LIN {X 0,Y 552.271,Z 509.997,A -85,B 0,C 180,E1 25736.055,E2 25736.055} C_VEL
LIN {X 0,Y 552.344,Z 509.997,A -85,B 0,C 180,E1 25732.825,E2 25732.825} C_VEL
LIN {X 0,Y 552.282,Z 509.996,A -85,B 0,C 180,E1 25729.569,E2 25729.569} C_VEL
LIN {X 0,Y 552.302,Z 509.994,A -85,B 0,C 180,E1 25726.174,E2 25726.174} C_VEL
LIN {X 0,Y 552.314,Z 509.999,A -85,B 0,C 180,E1 25723.054,E2 25723.054} C_VEL
LIN {X 0,Y 552.293,Z 509.995,A -85,B 0,C 180,E1 25719.77,E2 25719.77} C_VEL
LIN {X 0,Y 552.346,Z 509.995,A -85,B 0,C 180,E1 25716.531,E2 25716.531} C_VEL
LIN {X 0,Y 552.294,Z 509.997,A -85,B 0,C 180,E1 25713.322,E2 25713.322} C_VEL
LIN {X 0,Y 552.334,Z 509.997,A -85,B 0,C 180,E1 25712.64,E2 25712.64} C_VEL
LIN {X 0,Y 551.383,Z 510.118,A -85,B 0,C 180,E1 25711.84,E2 25711.84} C_VEL
LIN {X 0,Y 544.892,Z 510.92,A -85,B 0,C 180,E1 25709.597,E2 25709.597} C_VEL
LIN {X 0,Y 544.366,Z 510.988,A -85,B 0,C 180,E1 25709.012,E2 25709.012} C_VEL
LIN {X 0,Y 544.378,Z 510.984,A -85,B 0,C 180,E1 25705.546,E2 25705.546} C_VEL
LIN {X 0,Y 544.404,Z 510.987,A -85,B 0,C 180,E1 25702.162,E2 25702.162} C_VEL
LIN {X 0,Y 544.392,Z 511.152,A -85,B 0,C 180,E1 25698.937,E2 25698.937} C_VEL
LIN {X 0,Y 547.447,Z 523.021,A -85,B 0,C 180,E1 25697.272,E2 25697.272} C_VEL
LIN {X 0,Y 546.534,Z 551.773,A -85,B 0,C 180,E1 25693.828,E2 25693.828} C_VEL
LIN {X 0,Y 545.828,Z 580.978,A -85,B 0,C 180,E1 25690.42,E2 25690.42} C_VEL
LIN {X 0,Y 545.2,Z 610.398,A -85,B 0,C 180,E1 25687.05,E2 25687.05} C_VEL
LIN {X 0,Y 544.844,Z 632.663,A -85,B 0,C 180,E1 25684.588,E2 25684.588} C_VEL
LIN {X 0,Y 545.702,Z 641.313,A -85,B 0,C 180,E1 25684.418,E2 25684.418} C_VEL
LIN {X 0,Y 545.321,Z 744.483,A -85,B 0,C 180,E1 25683.029,E2 25683.029} C_VEL
LIN {X 0,Y 545.211,Z 758.833,A -85,B 0,C 180,E1 25682.65,E2 25682.65} C_VEL
LIN {X 0,Y 545.008,Z 773.495,A -85,B 0,C 180,E1 25682.051,E2 25682.051} C_VEL
LIN {X 0,Y 544.775,Z 786.249,A -85,B 0,C 180,E1 25681.334,E2 25681.334} C_VEL
LIN {X 0,Y 544.529,Z 799.172,A -85,B 0,C 180,E1 25680.385,E2 25680.385} C_VEL
LIN {X 0,Y 544.328,Z 811.081,A -85,B 0,C 180,E1 25679.245,E2 25679.245} C_VEL
LIN {X 0,Y 544.163,Z 820.825,A -85,B 0,C 180,E1 25678.055,E2 25678.055} C_VEL
LIN {X 0,Y 544.035,Z 829.383,A -85,B 0,C 180,E1 25676.721,E2 25676.721} C_VEL
LIN {X 0,Y 543.965,Z 836.569,A -85,B 0,C 180,E1 25675.238,E2 25675.238} C_VEL
LIN {X 0,Y 543.929,Z 841.752,A -85,B 0,C 180,E1 25673.732,E2 25673.732} C_VEL
LIN {X 0,Y 543.919,Z 845.089,A -85,B 0,C 180,E1 25672.248,E2 25672.248} C_VEL
LIN {X 0,Y 543.918,Z 846.806,A -85,B 0,C 180,E1 25670.662,E2 25670.662} C_VEL
LIN {X 0,Y 543.915,Z 846.71,A -85,B 0,C 180,E1 25669.096,E2 25669.096} C_VEL
LIN {X 0,Y 543.919,Z 844.892,A -85,B 0,C 180,E1 25667.543,E2 25667.543} C_VEL
LIN {X 0,Y 543.934,Z 840.933,A -85,B 0,C 180,E1 25665.893,E2 25665.893} C_VEL
LIN {X 0,Y 543.977,Z 835.236,A -85,B 0,C 180,E1 25664.365,E2 25664.365} C_VEL
LIN {X 0,Y 544.044,Z 828.675,A -85,B 0,C 180,E1 25663.062,E2 25663.062} C_VEL
LIN {X 0,Y 544.186,Z 819.39,A -85,B 0,C 180,E1 25661.658,E2 25661.658} C_VEL
LIN {X 0,Y 544.369,Z 808.765,A -85,B 0,C 180,E1 25660.421,E2 25660.421} C_VEL
LIN {X 0,Y 544.567,Z 797.66,A -85,B 0,C 180,E1 25659.403,E2 25659.403} C_VEL
LIN {X 0,Y 544.807,Z 784.989,A -85,B 0,C 180,E1 25658.494,E2 25658.494} C_VEL
LIN {X 0,Y 545.046,Z 771.112,A -85,B 0,C 180,E1 25657.747,E2 25657.747} C_VEL
LIN {X 0,Y 545.236,Z 756.981,A -85,B 0,C 180,E1 25657.202,E2 25657.202} C_VEL
LIN {X 0,Y 545.376,Z 741.93,A -85,B 0,C 180,E1 25656.832,E2 25656.832} C_VEL
LIN {X 0,Y 545.48,Z 637.399,A -85,B 0,C 180,E1 25655.434,E2 25655.434} C_VEL
LIN {X 0,Y 544.882,Z 632.555,A -85,B 0,C 180,E1 25655.315,E2 25655.315} C_VEL
LIN {X 0,Y 545.289,Z 602.715,A -85,B 0,C 180,E1 25651.995,E2 25651.995} C_VEL
LIN {X 0,Y 545.985,Z 572.64,A -85,B 0,C 180,E1 25648.53,E2 25648.53} C_VEL
LIN {X 0,Y 546.649,Z 544.661,A -85,B 0,C 180,E1 25645.278,E2 25645.278} C_VEL
LIN {X 0,Y 547.279,Z 522.265,A -85,B 0,C 180,E1 25642.599,E2 25642.599} C_VEL
LIN {X 0,Y 544.347,Z 511.079,A -85,B 0,C 180,E1 25640.991,E2 25640.991} C_VEL
LIN {X 0,Y 544.371,Z 510.988,A -85,B 0,C 180,E1 25637.806,E2 25637.806} C_VEL
LIN {X 0,Y 544.322,Z 510.99,A -85,B 0,C 180,E1 25634.553,E2 25634.553} C_VEL
LIN {X 0,Y 544.393,Z 510.99,A -85,B 0,C 180,E1 25631.363,E2 25631.363} C_VEL
LIN {X 0,Y 544.318,Z 510.989,A -85,B 0,C 180,E1 25628.22,E2 25628.22} C_VEL
LIN {X 0,Y 544.379,Z 510.983,A -85,B 0,C 180,E1 25625.012,E2 25625.012} C_VEL
LIN {X 0,Y 544.319,Z 510.989,A -85,B 0,C 180,E1 25621.832,E2 25621.832} C_VEL
LIN {X 0,Y 544.334,Z 510.982,A -85,B 0,C 180,E1 25618.434,E2 25618.434} C_VEL
LIN {X 0,Y 544.336,Z 510.989,A -85,B 0,C 180,E1 25615.377,E2 25615.377} C_VEL
LIN {X 0,Y 544.323,Z 510.987,A -85,B 0,C 180,E1 25612.002,E2 25612.002} C_VEL
LIN {X 0,Y 544.354,Z 510.99,A -85,B 0,C 180,E1 25609.019,E2 25609.019} C_VEL
LIN {X 0,Y 544.323,Z 510.988,A -85,B 0,C 180,E1 25605.735,E2 25605.735} C_VEL
LIN {X 0,Y 544.393,Z 510.985,A -85,B 0,C 180,E1 25602.524,E2 25602.524} C_VEL
LIN {X 0,Y 544.325,Z 510.986,A -85,B 0,C 180,E1 25599.326,E2 25599.326} C_VEL
LIN {X 0,Y 544.383,Z 510.983,A -85,B 0,C 180,E1 25596.09,E2 25596.09} C_VEL
LIN {X 0,Y 544.33,Z 510.982,A -85,B 0,C 180,E1 25592.937,E2 25592.937} C_VEL
LIN {X 0,Y 544.353,Z 510.986,A -85,B 0,C 180,E1 25589.61,E2 25589.61} C_VEL
LIN {X 0,Y 544.346,Z 510.982,A -85,B 0,C 180,E1 25586.56,E2 25586.56} C_VEL
LIN {X 0,Y 544.338,Z 510.986,A -85,B 0,C 180,E1 25583.147,E2 25583.147} C_VEL
LIN {X 0,Y 544.386,Z 510.988,A -85,B 0,C 180,E1 25579.976,E2 25579.976} C_VEL
LIN {X 0,Y 544.334,Z 510.979,A -85,B 0,C 180,E1 25576.762,E2 25576.762} C_VEL
LIN {X 0,Y 544.404,Z 510.987,A -85,B 0,C 180,E1 25573.597,E2 25573.597} C_VEL
LIN {X 0,Y 544.338,Z 510.983,A -85,B 0,C 180,E1 25570.371,E2 25570.371} C_VEL
LIN {X 0,Y 544.381,Z 510.981,A -85,B 0,C 180,E1 25567.069,E2 25567.069} C_VEL
LIN {X 0,Y 544.355,Z 510.987,A -85,B 0,C 180,E1 25563.897,E2 25563.897} C_VEL
LIN {X 0,Y 544.346,Z 510.974,A -85,B 0,C 180,E1 25560.421,E2 25560.421} C_VEL
LIN {X 0,Y 544.403,Z 510.988,A -85,B 0,C 180,E1 25557.158,E2 25557.158} C_VEL
LIN {X 0,Y 544.345,Z 510.984,A -85,B 0,C 180,E1 25553.885,E2 25553.885} C_VEL
LIN {X 0,Y 544.39,Z 510.982,A -85,B 0,C 180,E1 25550.592,E2 25550.592} C_VEL
LIN {X 0,Y 544.362,Z 510.987,A -85,B 0,C 180,E1 25547.375,E2 25547.375} C_VEL
LIN {X 0,Y 544.36,Z 510.981,A -85,B 0,C 180,E1 25544.008,E2 25544.008} C_VEL
LIN {X 0,Y 544.402,Z 510.985,A -85,B 0,C 180,E1 25540.728,E2 25540.728} C_VEL
LIN {X 0,Y 544.351,Z 510.984,A -85,B 0,C 180,E1 25537.425,E2 25537.425} C_VEL
LIN {X 0,Y 544.394,Z 510.977,A -85,B 0,C 180,E1 25534.08,E2 25534.08} C_VEL
LIN {X 0,Y 544.369,Z 510.987,A -85,B 0,C 180,E1 25530.874,E2 25530.874} C_VEL
LIN {X 0,Y 544.363,Z 510.983,A -85,B 0,C 180,E1 25527.441,E2 25527.441} C_VEL
LIN {X 0,Y 544.406,Z 510.985,A -85,B 0,C 180,E1 25524.135,E2 25524.135} C_VEL
LIN {X 0,Y 544.361,Z 510.984,A -85,B 0,C 180,E1 25520.811,E2 25520.811} C_VEL
LIN {X 0,Y 544.388,Z 510.982,A -85,B 0,C 180,E1 25517.431,E2 25517.431} C_VEL
LIN {X 0,Y 544.396,Z 510.987,A -85,B 0,C 180,E1 25514.1,E2 25514.1} C_VEL
LIN {X 0,Y 544.365,Z 510.985,A -85,B 0,C 180,E1 25510.823,E2 25510.823} C_VEL
LIN {X 0,Y 544.403,Z 510.987,A -85,B 0,C 180,E1 25507.57,E2 25507.57} C_VEL
LIN {X 0,Y 544.373,Z 510.989,A -85,B 0,C 180,E1 25504.195,E2 25504.195} C_VEL
LIN {X 0,Y 544.422,Z 511.233,A -85,B 0,C 180,E1 25502.897,E2 25502.897} C_VEL
LIN {X 0,Y 549.604,Z 527.102,A -85,B 0,C 180,E1 25501.29,E2 25501.29} C_VEL
LIN {X 0,Y 548.716,Z 570.56,A -85,B 0,C 180,E1 25498.124,E2 25498.124} C_VEL
LIN {X 0,Y 547.856,Z 611.744,A -85,B 0,C 180,E1 25495.147,E2 25495.147} C_VEL
LIN {X 0,Y 547.921,Z 615.465,A -85,B 0,C 180,E1 25494.922,E2 25494.922} C_VEL
LIN {X 0,Y 549.114,Z 624.911,A -85,B 0,C 180,E1 25494.729,E2 25494.729} C_VEL
LIN {X 0,Y 547.999,Z 824.349,A -85,B 0,C 180,E1 25491.964,E2 25491.964} C_VEL
LIN {X 0,Y 547.675,Z 843.385,A -85,B 0,C 180,E1 25491.502,E2 25491.502} C_VEL
LIN {X 0,Y 547.289,Z 861.41,A -85,B 0,C 180,E1 25490.87,E2 25490.87} C_VEL
LIN {X 0,Y 546.826,Z 879.05,A -85,B 0,C 180,E1 25490.049,E2 25490.049} C_VEL
LIN {X 0,Y 546.332,Z 895.775,A -85,B 0,C 180,E1 25489.067,E2 25489.067} C_VEL
LIN {X 0,Y 545.854,Z 911.628,A -85,B 0,C 180,E1 25487.922,E2 25487.922} C_VEL
LIN {X 0,Y 545.377,Z 926.557,A -85,B 0,C 180,E1 25486.618,E2 25486.618} C_VEL
LIN {X 0,Y 544.959,Z 940.217,A -85,B 0,C 180,E1 25485.187,E2 25485.187} C_VEL
LIN {X 0,Y 544.601,Z 952.914,A -85,B 0,C 180,E1 25483.592,E2 25483.592} C_VEL
LIN {X 0,Y 544.329,Z 964.228,A -85,B 0,C 180,E1 25481.872,E2 25481.872} C_VEL
LIN {X 0,Y 544.129,Z 973.992,A -85,B 0,C 180,E1 25480.054,E2 25480.054} C_VEL
LIN {X 0,Y 544.005,Z 982.175,A -85,B 0,C 180,E1 25478.137,E2 25478.137} C_VEL
LIN {X 0,Y 543.947,Z 988.41,A -85,B 0,C 180,E1 25476.227,E2 25476.227} C_VEL
LIN {X 0,Y 543.923,Z 992.876,A -85,B 0,C 180,E1 25474.323,E2 25474.323} C_VEL
LIN {X 0,Y 543.914,Z 995.792,A -85,B 0,C 180,E1 25472.319,E2 25472.319} C_VEL
LIN {X 0,Y 543.908,Z 996.939,A -85,B 0,C 180,E1 25470.317,E2 25470.317} C_VEL
LIN {X 0,Y 543.913,Z 996.348,A -85,B 0,C 180,E1 25468.316,E2 25468.316} C_VEL
LIN {X 0,Y 543.915,Z 994.005,A -85,B 0,C 180,E1 25466.313,E2 25466.313} C_VEL
LIN {X 0,Y 543.931,Z 990.101,A -85,B 0,C 180,E1 25464.411,E2 25464.411} C_VEL
LIN {X 0,Y 543.981,Z 984.474,A -85,B 0,C 180,E1 25462.503,E2 25462.503} C_VEL
LIN {X 0,Y 544.075,Z 977.436,A -85,B 0,C 180,E1 25460.695,E2 25460.695} C_VEL
LIN {X 0,Y 544.235,Z 968.529,A -85,B 0,C 180,E1 25458.88,E2 25458.88} C_VEL
LIN {X 0,Y 544.471,Z 958.168,A -85,B 0,C 180,E1 25457.164,E2 25457.164} C_VEL
LIN {X 0,Y 544.779,Z 946.371,A -85,B 0,C 180,E1 25455.548,E2 25455.548} C_VEL
LIN {X 0,Y 545.179,Z 933.106,A -85,B 0,C 180,E1 25454.035,E2 25454.035} C_VEL
LIN {X 0,Y 545.648,Z 918.253,A -85,B 0,C 180,E1 25452.624,E2 25452.624} C_VEL
LIN {X 0,Y 546.157,Z 902.275,A -85,B 0,C 180,E1 25451.373,E2 25451.373} C_VEL
LIN {X 0,Y 546.64,Z 885.106,A -85,B 0,C 180,E1 25450.28,E2 25450.28} C_VEL
LIN {X 0,Y 547.135,Z 867.88,A -85,B 0,C 180,E1 25449.407,E2 25449.407} C_VEL
LIN {X 0,Y 547.54,Z 849.631,A -85,B 0,C 180,E1 25448.695,E2 25448.695} C_VEL
LIN {X 0,Y 547.894,Z 830.962,A -85,B 0,C 180,E1 25448.175,E2 25448.175} C_VEL
LIN {X 0,Y 548.115,Z 810.606,A -85,B 0,C 180,E1 25447.822,E2 25447.822} C_VEL
LIN {X 0,Y 548.944,Z 622.019,A -85,B 0,C 180,E1 25445.222,E2 25445.222} C_VEL
LIN {X 0,Y 547.815,Z 614.387,A -85,B 0,C 180,E1 25445.038,E2 25445.038} C_VEL
LIN {X 0,Y 548.696,Z 571.729,A -85,B 0,C 180,E1 25441.961,E2 25441.961} C_VEL
LIN {X 0,Y 549.586,Z 527.86,A -85,B 0,C 180,E1 25438.767,E2 25438.767} C_VEL
LIN {X 0,Y 549.189,Z 525.155,A -85,B 0,C 180,E1 25438.534,E2 25438.534} C_VEL
LIN {X 0,Y 544.419,Z 511.228,A -85,B 0,C 180,E1 25437.106,E2 25437.106} C_VEL
LIN {X 0,Y 544.367,Z 510.99,A -85,B 0,C 180,E1 25433.739,E2 25433.739} C_VEL
LIN {X 0,Y 544.406,Z 510.984,A -85,B 0,C 180,E1 25430.415,E2 25430.415} C_VEL
LIN {X 0,Y 544.358,Z 510.985,A -85,B 0,C 180,E1 25427.127,E2 25427.127} C_VEL
LIN {X 0,Y 544.38,Z 510.99,A -85,B 0,C 180,E1 25423.802,E2 25423.802} C_VEL
LIN {X 0,Y 544.386,Z 510.984,A -85,B 0,C 180,E1 25420.51,E2 25420.51} C_VEL
LIN {X 0,Y 544.345,Z 510.988,A -85,B 0,C 180,E1 25417.148,E2 25417.148} C_VEL
LIN {X 0,Y 544.402,Z 510.987,A -85,B 0,C 180,E1 25413.896,E2 25413.896} C_VEL
LIN {X 0,Y 544.341,Z 510.986,A -85,B 0,C 180,E1 25410.706,E2 25410.706} C_VEL
LIN {X 0,Y 544.359,Z 510.988,A -85,B 0,C 180,E1 25407.335,E2 25407.335} C_VEL
LIN {X 0,Y 544.355,Z 510.986,A -85,B 0,C 180,E1 25404.18,E2 25404.18} C_VEL
LIN {X 0,Y 544.331,Z 510.988,A -85,B 0,C 180,E1 25400.876,E2 25400.876} C_VEL
LIN {X 0,Y 544.39,Z 510.985,A -85,B 0,C 180,E1 25397.641,E2 25397.641} C_VEL
LIN {X 0,Y 544.317,Z 510.983,A -85,B 0,C 180,E1 25394.467,E2 25394.467} C_VEL
LIN {X 0,Y 544.377,Z 510.987,A -85,B 0,C 180,E1 25391.226,E2 25391.226} C_VEL
LIN {X 0,Y 544.324,Z 510.988,A -85,B 0,C 180,E1 25388.025,E2 25388.025} C_VEL
LIN {X 0,Y 544.338,Z 510.984,A -85,B 0,C 180,E1 25384.636,E2 25384.636} C_VEL
LIN {X 0,Y 544.35,Z 510.989,A -85,B 0,C 180,E1 25381.579,E2 25381.579} C_VEL
LIN {X 0,Y 544.333,Z 510.987,A -85,B 0,C 180,E1 25378.21,E2 25378.21} C_VEL
LIN {X 0,Y 544.399,Z 510.982,A -85,B 0,C 180,E1 25374.942,E2 25374.942} C_VEL
LIN {X 0,Y 544.337,Z 510.987,A -85,B 0,C 180,E1 25371.762,E2 25371.762} C_VEL
LIN {X 0,Y 544.383,Z 510.985,A -85,B 0,C 180,E1 25368.451,E2 25368.451} C_VEL
LIN {X 0,Y 544.355,Z 510.985,A -85,B 0,C 180,E1 25365.316,E2 25365.316} C_VEL
LIN {X 0,Y 544.358,Z 510.984,A -85,B 0,C 180,E1 25361.916,E2 25361.916} C_VEL
LIN {X 0,Y 544.405,Z 510.984,A -85,B 0,C 180,E1 25358.6,E2 25358.6} C_VEL
LIN {X 0,Y 544.353,Z 510.983,A -85,B 0,C 180,E1 25355.358,E2 25355.358} C_VEL
LIN {X 0,Y 544.404,Z 510.983,A -85,B 0,C 180,E1 25352.044,E2 25352.044} C_VEL
LIN {X 0,Y 544.366,Z 510.988,A -85,B 0,C 180,E1 25349.012,E2 25349.012} C_VEL
LIN {X 0,Y 543.401,Z 511.113,A -85,B 0,C 180,E1 25348.201,E2 25348.201} C_VEL
LIN {X 0,Y 536.881,Z 511.92,A -85,B 0,C 180,E1 25345.865,E2 25345.865} C_VEL
LIN {X 0,Y 536.428,Z 511.975,A -85,B 0,C 180,E1 25345.33,E2 25345.33} C_VEL
LIN {X 0,Y 536.464,Z 511.977,A -85,B 0,C 180,E1 25342.026,E2 25342.026} C_VEL
LIN {X 0,Y 536.478,Z 512.244,A -85,B 0,C 180,E1 25339.304,E2 25339.304} C_VEL
LIN {X 0,Y 539.943,Z 525.069,A -85,B 0,C 180,E1 25337.47,E2 25337.47} C_VEL
LIN {X 0,Y 538.944,Z 553.767,A -85,B 0,C 180,E1 25333.996,E2 25333.996} C_VEL
LIN {X 0,Y 538.16,Z 583.042,A -85,B 0,C 180,E1 25330.545,E2 25330.545} C_VEL
LIN {X 0,Y 537.38,Z 612.981,A -85,B 0,C 180,E1 25327.04,E2 25327.04} C_VEL
LIN {X 0,Y 536.989,Z 632.746,A -85,B 0,C 180,E1 25324.801,E2 25324.801} C_VEL
LIN {X 0,Y 537.953,Z 642.099,A -85,B 0,C 180,E1 25324.62,E2 25324.62} C_VEL
LIN {X 0,Y 537.526,Z 744.402,A -85,B 0,C 180,E1 25323.223,E2 25323.223} C_VEL
LIN {X 0,Y 537.391,Z 759.339,A -85,B 0,C 180,E1 25322.821,E2 25322.821} C_VEL
LIN {X 0,Y 537.159,Z 774.098,A -85,B 0,C 180,E1 25322.201,E2 25322.201} C_VEL
LIN {X 0,Y 536.878,Z 787.415,A -85,B 0,C 180,E1 25321.426,E2 25321.426} C_VEL
LIN {X 0,Y 536.618,Z 799.477,A -85,B 0,C 180,E1 25320.513,E2 25320.513} C_VEL
LIN {X 0,Y 536.387,Z 811.37,A -85,B 0,C 180,E1 25319.353,E2 25319.353} C_VEL
LIN {X 0,Y 536.194,Z 821.279,A -85,B 0,C 180,E1 25318.112,E2 25318.112} C_VEL
LIN {X 0,Y 536.056,Z 829.352,A -85,B 0,C 180,E1 25316.828,E2 25316.828} C_VEL
LIN {X 0,Y 535.971,Z 836.696,A -85,B 0,C 180,E1 25315.286,E2 25315.286} C_VEL
LIN {X 0,Y 535.931,Z 841.829,A -85,B 0,C 180,E1 25313.761,E2 25313.761} C_VEL
LIN {X 0,Y 535.919,Z 845.135,A -85,B 0,C 180,E1 25312.252,E2 25312.252} C_VEL
LIN {X 0,Y 535.918,Z 846.824,A -85,B 0,C 180,E1 25310.644,E2 25310.644} C_VEL
LIN {X 0,Y 535.915,Z 846.691,A -85,B 0,C 180,E1 25309.053,E2 25309.053} C_VEL
LIN {X 0,Y 535.919,Z 844.836,A -85,B 0,C 180,E1 25307.477,E2 25307.477} C_VEL
LIN {X 0,Y 535.938,Z 840.849,A -85,B 0,C 180,E1 25305.803,E2 25305.803} C_VEL
LIN {X 0,Y 535.987,Z 835.114,A -85,B 0,C 180,E1 25304.252,E2 25304.252} C_VEL
LIN {X 0,Y 536.08,Z 827.859,A -85,B 0,C 180,E1 25302.821,E2 25302.821} C_VEL
LIN {X 0,Y 536.235,Z 819.186,A -85,B 0,C 180,E1 25301.506,E2 25301.506} C_VEL
LIN {X 0,Y 536.452,Z 808.273,A -85,B 0,C 180,E1 25300.227,E2 25300.227} C_VEL
LIN {X 0,Y 536.682,Z 796.645,A -85,B 0,C 180,E1 25299.164,E2 25299.164} C_VEL
LIN {X 0,Y 536.952,Z 784.539,A -85,B 0,C 180,E1 25298.295,E2 25298.295} C_VEL
LIN {X 0,Y 537.22,Z 770.517,A -85,B 0,C 180,E1 25297.538,E2 25297.538} C_VEL
LIN {X 0,Y 537.439,Z 756.126,A -85,B 0,C 180,E1 25296.987,E2 25296.987} C_VEL
LIN {X 0,Y 537.587,Z 741.359,A -85,B 0,C 180,E1 25296.629,E2 25296.629} C_VEL
LIN {X 0,Y 537.745,Z 638.26,A -85,B 0,C 180,E1 25295.232,E2 25295.232} C_VEL
LIN {X 0,Y 537.021,Z 632.585,A -85,B 0,C 180,E1 25295.099,E2 25295.099} C_VEL
LIN {X 0,Y 537.544,Z 603.794,A -85,B 0,C 180,E1 25291.811,E2 25291.811} C_VEL
LIN {X 0,Y 538.357,Z 572.84,A -85,B 0,C 180,E1 25288.19,E2 25288.19} C_VEL
LIN {X 0,Y 539.12,Z 544.837,A -85,B 0,C 180,E1 25284.892,E2 25284.892} C_VEL
LIN {X 0,Y 539.654,Z 524.364,A -85,B 0,C 180,E1 25282.412,E2 25282.412} C_VEL
LIN {X 0,Y 536.398,Z 512.075,A -85,B 0,C 180,E1 25280.613,E2 25280.613} C_VEL
LIN {X 0,Y 536.435,Z 511.979,A -85,B 0,C 180,E1 25277.294,E2 25277.294} C_VEL
LIN {X 0,Y 536.386,Z 511.979,A -85,B 0,C 180,E1 25274.208,E2 25274.208} C_VEL
LIN {X 0,Y 536.405,Z 511.977,A -85,B 0,C 180,E1 25270.849,E2 25270.849} C_VEL
LIN {X 0,Y 536.398,Z 511.978,A -85,B 0,C 180,E1 25267.766,E2 25267.766} C_VEL
LIN {X 0,Y 536.383,Z 511.978,A -85,B 0,C 180,E1 25264.377,E2 25264.377} C_VEL
LIN {X 0,Y 536.443,Z 511.969,A -85,B 0,C 180,E1 25261.137,E2 25261.137} C_VEL
LIN {X 0,Y 536.374,Z 511.97,A -85,B 0,C 180,E1 25257.91,E2 25257.91} C_VEL
LIN {X 0,Y 536.438,Z 511.977,A -85,B 0,C 180,E1 25254.706,E2 25254.706} C_VEL
LIN {X 0,Y 536.385,Z 511.976,A -85,B 0,C 180,E1 25251.496,E2 25251.496} C_VEL
LIN {X 0,Y 536.396,Z 511.972,A -85,B 0,C 180,E1 25248.052,E2 25248.052} C_VEL
LIN {X 0,Y 536.416,Z 511.977,A -85,B 0,C 180,E1 25244.906,E2 25244.906} C_VEL
LIN {X 0,Y 536.385,Z 511.97,A -85,B 0,C 180,E1 25241.576,E2 25241.576} C_VEL
LIN {X 0,Y 536.461,Z 511.977,A -85,B 0,C 180,E1 25238.364,E2 25238.364} C_VEL
LIN {X 0,Y 536.388,Z 511.973,A -85,B 0,C 180,E1 25235.088,E2 25235.088} C_VEL
LIN {X 0,Y 536.418,Z 511.975,A -85,B 0,C 180,E1 25231.711,E2 25231.711} C_VEL
LIN {X 0,Y 536.405,Z 511.977,A -85,B 0,C 180,E1 25228.624,E2 25228.624} C_VEL
LIN {X 0,Y 536.396,Z 511.969,A -85,B 0,C 180,E1 25225.151,E2 25225.151} C_VEL
LIN {X 0,Y 536.465,Z 511.977,A -85,B 0,C 180,E1 25221.886,E2 25221.886} C_VEL
LIN {X 0,Y 536.396,Z 511.97,A -85,B 0,C 180,E1 25218.588,E2 25218.588} C_VEL
LIN {X 0,Y 536.428,Z 511.973,A -85,B 0,C 180,E1 25215.237,E2 25215.237} C_VEL
LIN {X 0,Y 536.418,Z 511.977,A -85,B 0,C 180,E1 25212.05,E2 25212.05} C_VEL
LIN {X 0,Y 536.405,Z 511.963,A -85,B 0,C 180,E1 25208.684,E2 25208.684} C_VEL
LIN {X 0,Y 536.46,Z 511.976,A -85,B 0,C 180,E1 25205.455,E2 25205.455} C_VEL
LIN {X 0,Y 536.403,Z 511.972,A -85,B 0,C 180,E1 25202.137,E2 25202.137} C_VEL
LIN {X 0,Y 536.447,Z 511.97,A -85,B 0,C 180,E1 25198.825,E2 25198.825} C_VEL
LIN {X 0,Y 536.42,Z 511.977,A -85,B 0,C 180,E1 25195.617,E2 25195.617} C_VEL
LIN {X 0,Y 536.412,Z 511.965,A -85,B 0,C 180,E1 25192.18,E2 25192.18} C_VEL
LIN {X 0,Y 536.464,Z 511.977,A -85,B 0,C 180,E1 25188.932,E2 25188.932} C_VEL
LIN {X 0,Y 536.411,Z 511.969,A -85,B 0,C 180,E1 25185.646,E2 25185.646} C_VEL
LIN {X 0,Y 536.453,Z 511.972,A -85,B 0,C 180,E1 25182.314,E2 25182.314} C_VEL
LIN {X 0,Y 536.433,Z 511.973,A -85,B 0,C 180,E1 25179.028,E2 25179.028} C_VEL
LIN {X 0,Y 536.42,Z 511.973,A -85,B 0,C 180,E1 25175.674,E2 25175.674} C_VEL
LIN {X 0,Y 536.468,Z 511.974,A -85,B 0,C 180,E1 25172.349,E2 25172.349} C_VEL
LIN {X 0,Y 536.421,Z 511.973,A -85,B 0,C 180,E1 25169.022,E2 25169.022} C_VEL
LIN {X 0,Y 536.439,Z 511.97,A -85,B 0,C 180,E1 25165.615,E2 25165.615} C_VEL
LIN {X 0,Y 536.46,Z 511.978,A -85,B 0,C 180,E1 25162.314,E2 25162.314} C_VEL
LIN {X 0,Y 536.422,Z 511.974,A -85,B 0,C 180,E1 25158.996,E2 25158.996} C_VEL
LIN {X 0,Y 536.465,Z 511.969,A -85,B 0,C 180,E1 25155.66,E2 25155.66} C_VEL
LIN {X 0,Y 536.439,Z 511.976,A -85,B 0,C 180,E1 25152.272,E2 25152.272} C_VEL
LIN {X 0,Y 536.43,Z 511.974,A -85,B 0,C 180,E1 25148.82,E2 25148.82} C_VEL
LIN {X 0,Y 536.464,Z 511.973,A -85,B 0,C 180,E1 25145.423,E2 25145.423} C_VEL
LIN {X 0,Y 536.497,Z 512.203,A -85,B 0,C 180,E1 25143.331,E2 25143.331} C_VEL
LIN {X 0,Y 542.287,Z 529.764,A -85,B 0,C 180,E1 25141.513,E2 25141.513} C_VEL
LIN {X 0,Y 541.221,Z 573.376,A -85,B 0,C 180,E1 25138.284,E2 25138.284} C_VEL
LIN {X 0,Y 540.42,Z 615.037,A -85,B 0,C 180,E1 25135.298,E2 25135.298} C_VEL
LIN {X 0,Y 541.842,Z 625.928,A -85,B 0,C 180,E1 25135.069,E2 25135.069} C_VEL
LIN {X 0,Y 540.578,Z 824.349,A -85,B 0,C 180,E1 25132.282,E2 25132.282} C_VEL
LIN {X 0,Y 540.217,Z 843.359,A -85,B 0,C 180,E1 25131.815,E2 25131.815} C_VEL
LIN {X 0,Y 539.775,Z 861.408,A -85,B 0,C 180,E1 25131.174,E2 25131.174} C_VEL
LIN {X 0,Y 539.254,Z 879.047,A -85,B 0,C 180,E1 25130.343,E2 25130.343} C_VEL
LIN {X 0,Y 538.689,Z 895.773,A -85,B 0,C 180,E1 25129.348,E2 25129.348} C_VEL
LIN {X 0,Y 538.124,Z 912.195,A -85,B 0,C 180,E1 25128.141,E2 25128.141} C_VEL
LIN {X 0,Y 537.582,Z 927.111,A -85,B 0,C 180,E1 25126.811,E2 25126.811} C_VEL
LIN {X 0,Y 537.097,Z 940.945,A -85,B 0,C 180,E1 25125.328,E2 25125.328} C_VEL
LIN {X 0,Y 536.688,Z 953.683,A -85,B 0,C 180,E1 25123.686,E2 25123.686} C_VEL
LIN {X 0,Y 536.38,Z 964.863,A -85,B 0,C 180,E1 25121.942,E2 25121.942} C_VEL
LIN {X 0,Y 536.155,Z 974.506,A -85,B 0,C 180,E1 25120.096,E2 25120.096} C_VEL
LIN {X 0,Y 536.023,Z 982.174,A -85,B 0,C 180,E1 25118.259,E2 25118.259} C_VEL
LIN {X 0,Y 535.953,Z 988.411,A -85,B 0,C 180,E1 25116.32,E2 25116.32} C_VEL
LIN {X 0,Y 535.924,Z 992.876,A -85,B 0,C 180,E1 25114.388,E2 25114.388} C_VEL
LIN {X 0,Y 535.913,Z 995.792,A -85,B 0,C 180,E1 25112.354,E2 25112.354} C_VEL
LIN {X 0,Y 535.908,Z 996.939,A -85,B 0,C 180,E1 25110.322,E2 25110.322} C_VEL
LIN {X 0,Y 535.913,Z 996.348,A -85,B 0,C 180,E1 25108.291,E2 25108.291} C_VEL
LIN {X 0,Y 535.917,Z 994.004,A -85,B 0,C 180,E1 25106.258,E2 25106.258} C_VEL
LIN {X 0,Y 535.934,Z 990.101,A -85,B 0,C 180,E1 25104.327,E2 25104.327} C_VEL
LIN {X 0,Y 535.995,Z 984.474,A -85,B 0,C 180,E1 25102.391,E2 25102.391} C_VEL
LIN {X 0,Y 536.1,Z 977.436,A -85,B 0,C 180,E1 25100.556,E2 25100.556} C_VEL
LIN {X 0,Y 536.288,Z 968.53,A -85,B 0,C 180,E1 25098.713,E2 25098.713} C_VEL
LIN {X 0,Y 536.561,Z 958.169,A -85,B 0,C 180,E1 25096.971,E2 25096.971} C_VEL
LIN {X 0,Y 536.916,Z 946.371,A -85,B 0,C 180,E1 25095.332,E2 25095.332} C_VEL
LIN {X 0,Y 537.393,Z 932.684,A -85,B 0,C 180,E1 25093.751,E2 25093.751} C_VEL
LIN {X 0,Y 537.941,Z 917.637,A -85,B 0,C 180,E1 25092.311,E2 25092.311} C_VEL
LIN {X 0,Y 538.518,Z 901.481,A -85,B 0,C 180,E1 25091.042,E2 25091.042} C_VEL
LIN {X 0,Y 539.06,Z 884.78,A -85,B 0,C 180,E1 25089.973,E2 25089.973} C_VEL
LIN {X 0,Y 539.602,Z 867.882,A -85,B 0,C 180,E1 25089.106,E2 25089.106} C_VEL
LIN {X 0,Y 540.061,Z 849.634,A -85,B 0,C 180,E1 25088.385,E2 25088.385} C_VEL
LIN {X 0,Y 540.459,Z 831.074,A -85,B 0,C 180,E1 25087.861,E2 25087.861} C_VEL
LIN {X 0,Y 540.709,Z 810.733,A -85,B 0,C 180,E1 25087.503,E2 25087.503} C_VEL
LIN {X 0,Y 541.698,Z 623.241,A -85,B 0,C 180,E1 25084.885,E2 25084.885} C_VEL
LIN {X 0,Y 540.369,Z 614.302,A -85,B 0,C 180,E1 25084.67,E2 25084.67} C_VEL
LIN {X 0,Y 541.305,Z 569.367,A -85,B 0,C 180,E1 25081.423,E2 25081.423} C_VEL
LIN {X 0,Y 542.299,Z 529.19,A -85,B 0,C 180,E1 25078.445,E2 25078.445} C_VEL
LIN {X 0,Y 536.507,Z 512.263,A -85,B 0,C 180,E1 25076.688,E2 25076.688} C_VEL
LIN {X 0,Y 536.466,Z 511.975,A -85,B 0,C 180,E1 25074.58,E2 25074.58} C_VEL
LIN {X 0,Y 536.424,Z 511.974,A -85,B 0,C 180,E1 25071.229,E2 25071.229} C_VEL
LIN {X 0,Y 536.43,Z 511.977,A -85,B 0,C 180,E1 25067.729,E2 25067.729} C_VEL
LIN {X 0,Y 536.463,Z 511.973,A -85,B 0,C 180,E1 25064.459,E2 25064.459} C_VEL
LIN {X 0,Y 536.411,Z 511.975,A -85,B 0,C 180,E1 25061.146,E2 25061.146} C_VEL
LIN {X 0,Y 536.45,Z 511.978,A -85,B 0,C 180,E1 25057.798,E2 25057.798} C_VEL
LIN {X 0,Y 536.421,Z 511.973,A -85,B 0,C 180,E1 25054.516,E2 25054.516} C_VEL
LIN {X 0,Y 536.403,Z 511.976,A -85,B 0,C 180,E1 25051.086,E2 25051.086} C_VEL
LIN {X 0,Y 536.463,Z 511.97,A -85,B 0,C 180,E1 25047.892,E2 25047.892} C_VEL
LIN {X 0,Y 536.392,Z 511.975,A -85,B 0,C 180,E1 25044.68,E2 25044.68} C_VEL
LIN {X 0,Y 536.442,Z 511.978,A -85,B 0,C 180,E1 25041.427,E2 25041.427} C_VEL
LIN {X 0,Y 536.393,Z 511.974,A -85,B 0,C 180,E1 25038.25,E2 25038.25} C_VEL
LIN {X 0,Y 536.389,Z 511.971,A -85,B 0,C 180,E1 25034.796,E2 25034.796} C_VEL
LIN {X 0,Y 536.429,Z 511.979,A -85,B 0,C 180,E1 25031.613,E2 25031.613} C_VEL
LIN {X 0,Y 536.378,Z 511.977,A -85,B 0,C 180,E1 25028.36,E2 25028.36} C_VEL
LIN {X 0,Y 536.45,Z 511.97,A -85,B 0,C 180,E1 25025.133,E2 25025.133} C_VEL
LIN {X 0,Y 536.39,Z 511.978,A -85,B 0,C 180,E1 25021.923,E2 25021.923} C_VEL
LIN {X 0,Y 536.41,Z 511.976,A -85,B 0,C 180,E1 25018.504,E2 25018.504} C_VEL
LIN {X 0,Y 536.43,Z 511.975,A -85,B 0,C 180,E1 25015.296,E2 25015.296} C_VEL
LIN {X 0,Y 536.4,Z 511.976,A -85,B 0,C 180,E1 25011.963,E2 25011.963} C_VEL
LIN {X 0,Y 536.466,Z 511.975,A -85,B 0,C 180,E1 25008.714,E2 25008.714} C_VEL
LIN {X 0,Y 536.411,Z 511.974,A -85,B 0,C 180,E1 25005.425,E2 25005.425} C_VEL
LIN {X 0,Y 536.423,Z 511.972,A -85,B 0,C 180,E1 25001.976,E2 25001.976} C_VEL
LIN {X 0,Y 536.462,Z 511.973,A -85,B 0,C 180,E1 24998.688,E2 24998.688} C_VEL
LIN {X 0,Y 536.414,Z 511.972,A -85,B 0,C 180,E1 24995.438,E2 24995.438} C_VEL
LIN {X 0,Y 536.465,Z 511.972,A -85,B 0,C 180,E1 24992.048,E2 24992.048} C_VEL
LIN {X 0,Y 536.455,Z 511.977,A -85,B 0,C 180,E1 24988.598,E2 24988.598} C_VEL
LIN {X 0,Y 536.428,Z 511.975,A -85,B 0,C 180,E1 24985.33,E2 24985.33} C_VEL
LIN {X 0,Y 535.437,Z 512.103,A -85,B 0,C 180,E1 24984.508,E2 24984.508} C_VEL
LIN {X 0,Y 528.98,Z 512.908,A -85,B 0,C 180,E1 24982.136,E2 24982.136} C_VEL
LIN {X 0,Y 528.516,Z 512.964,A -85,B 0,C 180,E1 24981.594,E2 24981.594} C_VEL
LIN {X 0,Y 528.569,Z 513.247,A -85,B 0,C 180,E1 24979.711,E2 24979.711} C_VEL
LIN {X 0,Y 532.433,Z 527.639,A -85,B 0,C 180,E1 24977.61,E2 24977.61} C_VEL
LIN {X 0,Y 531.357,Z 556.238,A -85,B 0,C 180,E1 24974.119,E2 24974.119} C_VEL
LIN {X 0,Y 530.477,Z 585.499,A -85,B 0,C 180,E1 24970.627,E2 24970.627} C_VEL
LIN {X 0,Y 529.631,Z 614.708,A -85,B 0,C 180,E1 24967.159,E2 24967.159} C_VEL
LIN {X 0,Y 529.25,Z 632.819,A -85,B 0,C 180,E1 24965.088,E2 24965.088} C_VEL
LIN {X 0,Y 530.36,Z 642.793,A -85,B 0,C 180,E1 24964.883,E2 24964.883} C_VEL
LIN {X 0,Y 529.797,Z 744.646,A -85,B 0,C 180,E1 24963.443,E2 24963.443} C_VEL
LIN {X 0,Y 529.634,Z 758.971,A -85,B 0,C 180,E1 24963.049,E2 24963.049} C_VEL
LIN {X 0,Y 529.363,Z 773.363,A -85,B 0,C 180,E1 24962.435,E2 24962.435} C_VEL
LIN {X 0,Y 529.039,Z 786.603,A -85,B 0,C 180,E1 24961.657,E2 24961.657} C_VEL
LIN {X 0,Y 528.722,Z 799.187,A -85,B 0,C 180,E1 24960.699,E2 24960.699} C_VEL
LIN {X 0,Y 528.457,Z 811.32,A -85,B 0,C 180,E1 24959.501,E2 24959.501} C_VEL
LIN {X 0,Y 528.235,Z 821.262,A -85,B 0,C 180,E1 24958.238,E2 24958.238} C_VEL
LIN {X 0,Y 528.075,Z 829.526,A -85,B 0,C 180,E1 24956.9,E2 24956.9} C_VEL
LIN {X 0,Y 527.979,Z 836.819,A -85,B 0,C 180,E1 24955.336,E2 24955.336} C_VEL
LIN {X 0,Y 527.931,Z 842.245,A -85,B 0,C 180,E1 24953.669,E2 24953.669} C_VEL
LIN {X 0,Y 527.921,Z 845.526,A -85,B 0,C 180,E1 24952.021,E2 24952.021} C_VEL
LIN {X 0,Y 527.919,Z 846.889,A -85,B 0,C 180,E1 24950.507,E2 24950.507} C_VEL
LIN {X 0,Y 527.916,Z 846.528,A -85,B 0,C 180,E1 24948.779,E2 24948.779} C_VEL
LIN {X 0,Y 527.921,Z 844.348,A -85,B 0,C 180,E1 24947.182,E2 24947.182} C_VEL
LIN {X 0,Y 527.944,Z 840.405,A -85,B 0,C 180,E1 24945.598,E2 24945.598} C_VEL
LIN {X 0,Y 528.006,Z 834.519,A -85,B 0,C 180,E1 24944.025,E2 24944.025} C_VEL
LIN {X 0,Y 528.12,Z 827.044,A -85,B 0,C 180,E1 24942.573,E2 24942.573} C_VEL
LIN {X 0,Y 528.306,Z 818.121,A -85,B 0,C 180,E1 24941.239,E2 24941.239} C_VEL
LIN {X 0,Y 528.555,Z 807.188,A -85,B 0,C 180,E1 24939.965,E2 24939.965} C_VEL
LIN {X 0,Y 528.829,Z 794.954,A -85,B 0,C 180,E1 24938.862,E2 24938.862} C_VEL
LIN {X 0,Y 529.171,Z 781.448,A -85,B 0,C 180,E1 24937.926,E2 24937.926} C_VEL
LIN {X 0,Y 529.468,Z 768.133,A -85,B 0,C 180,E1 24937.229,E2 24937.229} C_VEL
LIN {X 0,Y 529.726,Z 753.411,A -85,B 0,C 180,E1 24936.688,E2 24936.688} C_VEL
LIN {X 0,Y 529.877,Z 737.548,A -85,B 0,C 180,E1 24936.346,E2 24936.346} C_VEL
LIN {X 0,Y 530.136,Z 639.111,A -85,B 0,C 180,E1 24934.975,E2 24934.975} C_VEL
LIN {X 0,Y 529.246,Z 632.589,A -85,B 0,C 180,E1 24934.821,E2 24934.821} C_VEL
LIN {X 0,Y 529.818,Z 604.948,A -85,B 0,C 180,E1 24931.621,E2 24931.621} C_VEL
LIN {X 0,Y 530.699,Z 574.865,A -85,B 0,C 180,E1 24928.055,E2 24928.055} C_VEL
LIN {X 0,Y 531.562,Z 546.856,A -85,B 0,C 180,E1 24924.711,E2 24924.711} C_VEL
LIN {X 0,Y 532.272,Z 527.363,A -85,B 0,C 180,E1 24922.335,E2 24922.335} C_VEL
LIN {X 0,Y 528.477,Z 513.102,A -85,B 0,C 180,E1 24920.251,E2 24920.251} C_VEL
LIN {X 0,Y 528.451,Z 512.967,A -85,B 0,C 180,E1 24916.765,E2 24916.765} C_VEL
LIN {X 0,Y 528.503,Z 512.968,A -85,B 0,C 180,E1 24913.574,E2 24913.574} C_VEL
LIN {X 0,Y 528.443,Z 512.966,A -85,B 0,C 180,E1 24910.319,E2 24910.319} C_VEL
LIN {X 0,Y 528.5,Z 512.949,A -85,B 0,C 180,E1 24907.063,E2 24907.063} C_VEL
LIN {X 0,Y 528.446,Z 512.967,A -85,B 0,C 180,E1 24903.843,E2 24903.843} C_VEL
LIN {X 0,Y 528.449,Z 512.952,A -85,B 0,C 180,E1 24900.409,E2 24900.409} C_VEL
LIN {X 0,Y 528.476,Z 512.958,A -85,B 0,C 180,E1 24897.243,E2 24897.243} C_VEL
LIN {X 0,Y 528.439,Z 512.966,A -85,B 0,C 180,E1 24893.894,E2 24893.894} C_VEL
LIN {X 0,Y 528.519,Z 512.967,A -85,B 0,C 180,E1 24890.675,E2 24890.675} C_VEL
LIN {X 0,Y 528.443,Z 512.96,A -85,B 0,C 180,E1 24887.512,E2 24887.512} C_VEL
LIN {X 0,Y 528.481,Z 512.966,A -85,B 0,C 180,E1 24884.192,E2 24884.192} C_VEL
LIN {X 0,Y 528.456,Z 512.959,A -85,B 0,C 180,E1 24881.037,E2 24881.037} C_VEL
LIN {X 0,Y 528.454,Z 512.966,A -85,B 0,C 180,E1 24877.559,E2 24877.559} C_VEL
LIN {X 0,Y 528.521,Z 512.954,A -85,B 0,C 180,E1 24874.242,E2 24874.242} C_VEL
LIN {X 0,Y 528.452,Z 512.965,A -85,B 0,C 180,E1 24870.974,E2 24870.974} C_VEL
LIN {X 0,Y 528.484,Z 512.957,A -85,B 0,C 180,E1 24867.615,E2 24867.615} C_VEL
LIN {X 0,Y 528.47,Z 512.959,A -85,B 0,C 180,E1 24864.478,E2 24864.478} C_VEL
LIN {X 0,Y 528.461,Z 512.964,A -85,B 0,C 180,E1 24861.069,E2 24861.069} C_VEL
LIN {X 0,Y 528.523,Z 512.952,A -85,B 0,C 180,E1 24857.733,E2 24857.733} C_VEL
LIN {X 0,Y 528.46,Z 512.964,A -85,B 0,C 180,E1 24854.463,E2 24854.463} C_VEL
LIN {X 0,Y 528.492,Z 512.958,A -85,B 0,C 180,E1 24851.127,E2 24851.127} C_VEL
LIN {X 0,Y 528.478,Z 512.953,A -85,B 0,C 180,E1 24847.939,E2 24847.939} C_VEL
LIN {X 0,Y 528.469,Z 512.963,A -85,B 0,C 180,E1 24844.558,E2 24844.558} C_VEL
LIN {X 0,Y 528.524,Z 512.952,A -85,B 0,C 180,E1 24841.301,E2 24841.301} C_VEL
LIN {X 0,Y 528.466,Z 512.961,A -85,B 0,C 180,E1 24838.049,E2 24838.049} C_VEL
LIN {X 0,Y 528.507,Z 512.958,A -85,B 0,C 180,E1 24834.681,E2 24834.681} C_VEL
LIN {X 0,Y 528.488,Z 512.956,A -85,B 0,C 180,E1 24831.404,E2 24831.404} C_VEL
LIN {X 0,Y 528.473,Z 512.963,A -85,B 0,C 180,E1 24827.984,E2 24827.984} C_VEL
LIN {X 0,Y 528.53,Z 512.957,A -85,B 0,C 180,E1 24824.642,E2 24824.642} C_VEL
LIN {X 0,Y 528.479,Z 512.965,A -85,B 0,C 180,E1 24821.353,E2 24821.353} C_VEL
LIN {X 0,Y 528.488,Z 512.959,A -85,B 0,C 180,E1 24817.884,E2 24817.884} C_VEL
LIN {X 0,Y 528.524,Z 512.96,A -85,B 0,C 180,E1 24814.568,E2 24814.568} C_VEL
LIN {X 0,Y 528.476,Z 512.964,A -85,B 0,C 180,E1 24811.278,E2 24811.278} C_VEL
LIN {X 0,Y 528.524,Z 512.959,A -85,B 0,C 180,E1 24807.938,E2 24807.938} C_VEL
LIN {X 0,Y 528.509,Z 512.962,A -85,B 0,C 180,E1 24804.493,E2 24804.493} C_VEL
LIN {X 0,Y 528.482,Z 512.96,A -85,B 0,C 180,E1 24801.088,E2 24801.088} C_VEL
LIN {X 0,Y 528.525,Z 512.961,A -85,B 0,C 180,E1 24797.811,E2 24797.811} C_VEL
LIN {X 0,Y 528.494,Z 512.963,A -85,B 0,C 180,E1 24794.424,E2 24794.424} C_VEL
LIN {X 0,Y 528.491,Z 512.963,A -85,B 0,C 180,E1 24790.887,E2 24790.887} C_VEL
LIN {X 0,Y 528.525,Z 512.965,A -85,B 0,C 180,E1 24787.526,E2 24787.526} C_VEL
LIN {X 0,Y 528.496,Z 512.968,A -85,B 0,C 180,E1 24784.185,E2 24784.185} C_VEL
LIN {X 0,Y 528.589,Z 513.411,A -85,B 0,C 180,E1 24783.733,E2 24783.733} C_VEL
LIN {X 0,Y 534.978,Z 532.365,A -85,B 0,C 180,E1 24781.747,E2 24781.747} C_VEL
LIN {X 0,Y 533.768,Z 574.446,A -85,B 0,C 180,E1 24778.578,E2 24778.578} C_VEL
LIN {X 0,Y 532.811,Z 615.221,A -85,B 0,C 180,E1 24775.598,E2 24775.598} C_VEL
LIN {X 0,Y 534.386,Z 626.877,A -85,B 0,C 180,E1 24775.368,E2 24775.368} C_VEL
LIN {X 0,Y 533.239,Z 818.243,A -85,B 0,C 180,E1 24772.713,E2 24772.713} C_VEL
LIN {X 0,Y 532.885,Z 837.746,A -85,B 0,C 180,E1 24772.294,E2 24772.294} C_VEL
LIN {X 0,Y 532.413,Z 856.435,A -85,B 0,C 180,E1 24771.684,E2 24771.684} C_VEL
LIN {X 0,Y 531.876,Z 874.402,A -85,B 0,C 180,E1 24770.885,E2 24770.885} C_VEL
LIN {X 0,Y 531.226,Z 891.453,A -85,B 0,C 180,E1 24769.917,E2 24769.917} C_VEL
LIN {X 0,Y 530.612,Z 907.79,A -85,B 0,C 180,E1 24768.766,E2 24768.766} C_VEL
LIN {X 0,Y 529.985,Z 923.085,A -85,B 0,C 180,E1 24767.455,E2 24767.455} C_VEL
LIN {X 0,Y 529.419,Z 937.247,A -85,B 0,C 180,E1 24765.993,E2 24765.993} C_VEL
LIN {X 0,Y 528.922,Z 950.574,A -85,B 0,C 180,E1 24764.338,E2 24764.338} C_VEL
LIN {X 0,Y 528.527,Z 962.316,A -85,B 0,C 180,E1 24762.566,E2 24762.566} C_VEL
LIN {X 0,Y 528.246,Z 972.445,A -85,B 0,C 180,E1 24760.69,E2 24760.69} C_VEL
LIN {X 0,Y 528.066,Z 980.555,A -85,B 0,C 180,E1 24758.823,E2 24758.823} C_VEL
LIN {X 0,Y 527.973,Z 987.198,A -85,B 0,C 180,E1 24756.853,E2 24756.853} C_VEL
LIN {X 0,Y 527.924,Z 992.049,A -85,B 0,C 180,E1 24754.89,E2 24754.89} C_VEL
LIN {X 0,Y 527.912,Z 995.224,A -85,B 0,C 180,E1 24752.932,E2 24752.932} C_VEL
LIN {X 0,Y 527.911,Z 996.826,A -85,B 0,C 180,E1 24750.869,E2 24750.869} C_VEL
LIN {X 0,Y 527.906,Z 996.685,A -85,B 0,C 180,E1 24748.808,E2 24748.808} C_VEL
LIN {X 0,Y 527.913,Z 994.956,A -85,B 0,C 180,E1 24746.853,E2 24746.853} C_VEL
LIN {X 0,Y 527.929,Z 991.369,A -85,B 0,C 180,E1 24744.786,E2 24744.786} C_VEL
LIN {X 0,Y 527.98,Z 986.239,A -85,B 0,C 180,E1 24742.822,E2 24742.822} C_VEL
LIN {X 0,Y 528.097,Z 979.27,A -85,B 0,C 180,E1 24740.851,E2 24740.851} C_VEL
LIN {X 0,Y 528.286,Z 970.822,A -85,B 0,C 180,E1 24738.982,E2 24738.982} C_VEL
LIN {X 0,Y 528.571,Z 960.971,A -85,B 0,C 180,E1 24737.216,E2 24737.216} C_VEL
LIN {X 0,Y 528.948,Z 949.751,A -85,B 0,C 180,E1 24735.554,E2 24735.554} C_VEL
LIN {X 0,Y 529.44,Z 936.652,A -85,B 0,C 180,E1 24733.941,E2 24733.941} C_VEL
LIN {X 0,Y 530.006,Z 922.506,A -85,B 0,C 180,E1 24732.491,E2 24732.491} C_VEL
LIN {X 0,Y 530.625,Z 907.427,A -85,B 0,C 180,E1 24731.206,E2 24731.206} C_VEL
LIN {X 0,Y 531.225,Z 891.494,A -85,B 0,C 180,E1 24730.085,E2 24730.085} C_VEL
LIN {X 0,Y 531.874,Z 874.405,A -85,B 0,C 180,E1 24729.115,E2 24729.115} C_VEL
LIN {X 0,Y 532.412,Z 856.508,A -85,B 0,C 180,E1 24728.319,E2 24728.319} C_VEL
LIN {X 0,Y 532.885,Z 837.666,A -85,B 0,C 180,E1 24727.703,E2 24727.703} C_VEL
LIN {X 0,Y 533.241,Z 818.094,A -85,B 0,C 180,E1 24727.285,E2 24727.285} C_VEL
LIN {X 0,Y 534.352,Z 631.084,A -85,B 0,C 180,E1 24724.693,E2 24724.693} C_VEL
LIN {X 0,Y 534.094,Z 623.444,A -85,B 0,C 180,E1 24724.576,E2 24724.576} C_VEL
LIN {X 0,Y 532.75,Z 614.39,A -85,B 0,C 180,E1 24724.371,E2 24724.371} C_VEL
LIN {X 0,Y 533.849,Z 571.134,A -85,B 0,C 180,E1 24721.176,E2 24721.176} C_VEL
LIN {X 0,Y 534.982,Z 531.997,A -85,B 0,C 180,E1 24718.227,E2 24718.227} C_VEL
LIN {X 0,Y 528.563,Z 513.274,A -85,B 0,C 180,E1 24716.248,E2 24716.248} C_VEL
LIN {X 0,Y 528.523,Z 512.965,A -85,B 0,C 180,E1 24714.765,E2 24714.765} C_VEL
LIN {X 0,Y 528.483,Z 512.964,A -85,B 0,C 180,E1 24711.372,E2 24711.372} C_VEL
LIN {X 0,Y 528.509,Z 512.967,A -85,B 0,C 180,E1 24707.961,E2 24707.961} C_VEL
LIN {X 0,Y 528.515,Z 512.962,A -85,B 0,C 180,E1 24704.577,E2 24704.577} C_VEL
LIN {X 0,Y 528.473,Z 512.965,A -85,B 0,C 180,E1 24701.178,E2 24701.178} C_VEL
LIN {X 0,Y 528.512,Z 512.966,A -85,B 0,C 180,E1 24697.803,E2 24697.803} C_VEL
LIN {X 0,Y 528.479,Z 512.962,A -85,B 0,C 180,E1 24694.582,E2 24694.582} C_VEL
LIN {X 0,Y 528.465,Z 512.965,A -85,B 0,C 180,E1 24691.099,E2 24691.099} C_VEL
LIN {X 0,Y 528.524,Z 512.959,A -85,B 0,C 180,E1 24687.857,E2 24687.857} C_VEL
LIN {X 0,Y 528.454,Z 512.964,A -85,B 0,C 180,E1 24684.598,E2 24684.598} C_VEL
LIN {X 0,Y 528.487,Z 512.967,A -85,B 0,C 180,E1 24681.3,E2 24681.3} C_VEL
LIN {X 0,Y 528.458,Z 512.962,A -85,B 0,C 180,E1 24678.191,E2 24678.191} C_VEL
LIN {X 0,Y 528.451,Z 512.959,A -85,B 0,C 180,E1 24674.799,E2 24674.799} C_VEL
LIN {X 0,Y 528.494,Z 512.968,A -85,B 0,C 180,E1 24671.568,E2 24671.568} C_VEL
LIN {X 0,Y 528.439,Z 512.966,A -85,B 0,C 180,E1 24668.268,E2 24668.268} C_VEL
LIN {X 0,Y 528.495,Z 512.959,A -85,B 0,C 180,E1 24664.992,E2 24664.992} C_VEL
LIN {X 0,Y 528.46,Z 512.967,A -85,B 0,C 180,E1 24661.735,E2 24661.735} C_VEL
LIN {X 0,Y 528.458,Z 512.965,A -85,B 0,C 180,E1 24658.265,E2 24658.265} C_VEL
LIN {X 0,Y 528.517,Z 512.959,A -85,B 0,C 180,E1 24655.007,E2 24655.007} C_VEL
LIN {X 0,Y 528.46,Z 512.965,A -85,B 0,C 180,E1 24651.732,E2 24651.732} C_VEL
LIN {X 0,Y 528.491,Z 512.963,A -85,B 0,C 180,E1 24648.32,E2 24648.32} C_VEL
LIN {X 0,Y 528.496,Z 512.963,A -85,B 0,C 180,E1 24645.09,E2 24645.09} C_VEL
LIN {X 0,Y 528.472,Z 512.962,A -85,B 0,C 180,E1 24641.695,E2 24641.695} C_VEL
LIN {X 0,Y 528.528,Z 512.962,A -85,B 0,C 180,E1 24638.352,E2 24638.352} C_VEL
LIN {X 0,Y 528.492,Z 512.963,A -85,B 0,C 180,E1 24634.975,E2 24634.975} C_VEL
LIN {X 0,Y 528.486,Z 512.964,A -85,B 0,C 180,E1 24631.525,E2 24631.525} C_VEL
LIN {X 0,Y 528.527,Z 512.961,A -85,B 0,C 180,E1 24628.27,E2 24628.27} C_VEL
LIN {X 0,Y 528.492,Z 512.967,A -85,B 0,C 180,E1 24624.89,E2 24624.89} C_VEL
LIN {X 0,Y 528.516,Z 512.964,A -85,B 0,C 180,E1 24621.594,E2 24621.594} C_VEL
LIN {X 0,Y 527.55,Z 513.373,A -85,B 0,C 180,E1 24621.023,E2 24621.023} C_VEL
LIN {X 0,Y 524.282,Z 515.426,A -85,B 0,C 180,E1 24620.191,E2 24620.191} C_VEL
LIN {X 0,Y 522.43,Z 517.953,A -85,B 0,C 180,E1 24619.614,E2 24619.614} C_VEL
LIN {X 0,Y 522.342,Z 520.404,A -85,B 0,C 180,E1 24619.199,E2 24619.199} C_VEL
LIN {X 0,Y 524.938,Z 530.311,A -85,B 0,C 180,E1 24617.75,E2 24617.75} C_VEL
LIN {X 0,Y 523.771,Z 558.768,A -85,B 0,C 180,E1 24614.238,E2 24614.238} C_VEL
LIN {X 0,Y 522.79,Z 588.047,A -85,B 0,C 180,E1 24610.7,E2 24610.7} C_VEL
LIN {X 0,Y 521.876,Z 616.67,A -85,B 0,C 180,E1 24607.254,E2 24607.254} C_VEL
LIN {X 0,Y 521.534,Z 632.755,A -85,B 0,C 180,E1 24605.406,E2 24605.406} C_VEL
LIN {X 0,Y 522.866,Z 643.44,A -85,B 0,C 180,E1 24605.182,E2 24605.182} C_VEL
LIN {X 0,Y 522.215,Z 745.259,A -85,B 0,C 180,E1 24603.714,E2 24603.714} C_VEL
LIN {X 0,Y 522.035,Z 759.752,A -85,B 0,C 180,E1 24603.308,E2 24603.308} C_VEL
LIN {X 0,Y 521.749,Z 773.719,A -85,B 0,C 180,E1 24602.707,E2 24602.707} C_VEL
LIN {X 0,Y 521.405,Z 786.591,A -85,B 0,C 180,E1 24601.951,E2 24601.951} C_VEL
LIN {X 0,Y 520.997,Z 799.53,A -85,B 0,C 180,E1 24600.948,E2 24600.948} C_VEL
LIN {X 0,Y 520.652,Z 811.169,A -85,B 0,C 180,E1 24599.77,E2 24599.77} C_VEL
LIN {X 0,Y 520.375,Z 820.452,A -85,B 0,C 180,E1 24598.579,E2 24598.579} C_VEL
LIN {X 0,Y 520.141,Z 829.307,A -85,B 0,C 180,E1 24597.124,E2 24597.124} C_VEL
LIN {X 0,Y 519.999,Z 836.616,A -85,B 0,C 180,E1 24595.509,E2 24595.509} C_VEL
LIN {X 0,Y 519.934,Z 842.005,A -85,B 0,C 180,E1 24593.815,E2 24593.815} C_VEL
LIN {X 0,Y 519.92,Z 845.226,A -85,B 0,C 180,E1 24592.259,E2 24592.259} C_VEL
LIN {X 0,Y 519.919,Z 846.86,A -85,B 0,C 180,E1 24590.602,E2 24590.602} C_VEL
LIN {X 0,Y 519.915,Z 846.602,A -85,B 0,C 180,E1 24588.883,E2 24588.883} C_VEL
LIN {X 0,Y 519.92,Z 844.722,A -85,B 0,C 180,E1 24587.339,E2 24587.339} C_VEL
LIN {X 0,Y 519.947,Z 840.698,A -85,B 0,C 180,E1 24585.615,E2 24585.615} C_VEL
LIN {X 0,Y 520.03,Z 834.591,A -85,B 0,C 180,E1 24583.904,E2 24583.904} C_VEL
LIN {X 0,Y 520.182,Z 827.288,A -85,B 0,C 180,E1 24582.429,E2 24582.429} C_VEL
LIN {X 0,Y 520.423,Z 818.553,A -85,B 0,C 180,E1 24581.074,E2 24581.074} C_VEL
LIN {X 0,Y 520.728,Z 808.371,A -85,B 0,C 180,E1 24579.837,E2 24579.837} C_VEL
LIN {X 0,Y 521.071,Z 796.511,A -85,B 0,C 180,E1 24578.717,E2 24578.717} C_VEL
LIN {X 0,Y 521.447,Z 784.312,A -85,B 0,C 180,E1 24577.823,E2 24577.823} C_VEL
LIN {X 0,Y 521.772,Z 771.366,A -85,B 0,C 180,E1 24577.098,E2 24577.098} C_VEL
LIN {X 0,Y 522.053,Z 757.107,A -85,B 0,C 180,E1 24576.528,E2 24576.528} C_VEL
LIN {X 0,Y 522.242,Z 742.309,A -85,B 0,C 180,E1 24576.151,E2 24576.151} C_VEL
LIN {X 0,Y 522.593,Z 639.875,A -85,B 0,C 180,E1 24574.689,E2 24574.689} C_VEL
LIN {X 0,Y 521.489,Z 632.38,A -85,B 0,C 180,E1 24574.507,E2 24574.507} C_VEL
LIN {X 0,Y 522.127,Z 605.184,A -85,B 0,C 180,E1 24571.315,E2 24571.315} C_VEL
LIN {X 0,Y 523.069,Z 575.978,A -85,B 0,C 180,E1 24567.808,E2 24567.808} C_VEL
LIN {X 0,Y 524.045,Z 547.982,A -85,B 0,C 180,E1 24564.415,E2 24564.415} C_VEL
LIN {X 0,Y 524.666,Z 529.433,A -85,B 0,C 180,E1 24562.113,E2 24562.113} C_VEL
LIN {X 0,Y 520.572,Z 514.075,A -85,B 0,C 180,E1 24559.85,E2 24559.85} C_VEL
LIN {X 0,Y 520.508,Z 513.956,A -85,B 0,C 180,E1 24556.559,E2 24556.559} C_VEL
LIN {X 0,Y 520.565,Z 513.954,A -85,B 0,C 180,E1 24553.255,E2 24553.255} C_VEL
LIN {X 0,Y 520.512,Z 513.954,A -85,B 0,C 180,E1 24550.006,E2 24550.006} C_VEL
LIN {X 0,Y 520.506,Z 513.936,A -85,B 0,C 180,E1 24546.45,E2 24546.45} C_VEL
LIN {X 0,Y 520.565,Z 513.956,A -85,B 0,C 180,E1 24543.169,E2 24543.169} C_VEL
LIN {X 0,Y 520.497,Z 513.939,A -85,B 0,C 180,E1 24539.91,E2 24539.91} C_VEL
LIN {X 0,Y 520.536,Z 513.956,A -85,B 0,C 180,E1 24536.547,E2 24536.547} C_VEL
LIN {X 0,Y 520.52,Z 513.955,A -85,B 0,C 180,E1 24533.318,E2 24533.318} C_VEL
LIN {X 0,Y 520.505,Z 513.956,A -85,B 0,C 180,E1 24529.866,E2 24529.866} C_VEL
LIN {X 0,Y 520.567,Z 513.947,A -85,B 0,C 180,E1 24526.713,E2 24526.713} C_VEL
LIN {X 0,Y 520.506,Z 513.955,A -85,B 0,C 180,E1 24523.442,E2 24523.442} C_VEL
LIN {X 0,Y 520.544,Z 513.952,A -85,B 0,C 180,E1 24520.051,E2 24520.051} C_VEL
LIN {X 0,Y 520.519,Z 513.956,A -85,B 0,C 180,E1 24516.959,E2 24516.959} C_VEL
LIN {X 0,Y 520.516,Z 513.946,A -85,B 0,C 180,E1 24513.456,E2 24513.456} C_VEL
LIN {X 0,Y 520.578,Z 513.956,A -85,B 0,C 180,E1 24510.203,E2 24510.203} C_VEL
LIN {X 0,Y 520.514,Z 513.946,A -85,B 0,C 180,E1 24506.958,E2 24506.958} C_VEL
LIN {X 0,Y 520.563,Z 513.952,A -85,B 0,C 180,E1 24503.633,E2 24503.633} C_VEL
LIN {X 0,Y 520.532,Z 513.954,A -85,B 0,C 180,E1 24500.395,E2 24500.395} C_VEL
LIN {X 0,Y 520.525,Z 513.943,A -85,B 0,C 180,E1 24496.956,E2 24496.956} C_VEL
LIN {X 0,Y 520.586,Z 513.955,A -85,B 0,C 180,E1 24493.643,E2 24493.643} C_VEL
LIN {X 0,Y 520.524,Z 513.949,A -85,B 0,C 180,E1 24490.291,E2 24490.291} C_VEL
LIN {X 0,Y 520.537,Z 513.948,A -85,B 0,C 180,E1 24486.783,E2 24486.783} C_VEL
LIN {X 0,Y 520.57,Z 513.955,A -85,B 0,C 180,E1 24483.524,E2 24483.524} C_VEL
LIN {X 0,Y 520.525,Z 513.938,A -85,B 0,C 180,E1 24480.22,E2 24480.22} C_VEL
LIN {X 0,Y 520.581,Z 513.951,A -85,B 0,C 180,E1 24476.917,E2 24476.917} C_VEL
LIN {X 0,Y 520.541,Z 513.951,A -85,B 0,C 180,E1 24473.604,E2 24473.604} C_VEL
LIN {X 0,Y 520.538,Z 513.95,A -85,B 0,C 180,E1 24470.157,E2 24470.157} C_VEL
LIN {X 0,Y 520.588,Z 513.946,A -85,B 0,C 180,E1 24466.788,E2 24466.788} C_VEL
LIN {X 0,Y 520.538,Z 513.95,A -85,B 0,C 180,E1 24463.421,E2 24463.421} C_VEL
LIN {X 0,Y 520.546,Z 513.946,A -85,B 0,C 180,E1 24459.89,E2 24459.89} C_VEL
LIN {X 0,Y 520.59,Z 513.954,A -85,B 0,C 180,E1 24456.574,E2 24456.574} C_VEL
LIN {X 0,Y 520.541,Z 513.946,A -85,B 0,C 180,E1 24453.167,E2 24453.167} C_VEL
LIN {X 0,Y 520.566,Z 513.947,A -85,B 0,C 180,E1 24449.786,E2 24449.786} C_VEL
LIN {X 0,Y 520.579,Z 513.956,A -85,B 0,C 180,E1 24446.417,E2 24446.417} C_VEL
LIN {X 0,Y 520.543,Z 513.952,A -85,B 0,C 180,E1 24443.035,E2 24443.035} C_VEL
LIN {X 0,Y 520.59,Z 513.949,A -85,B 0,C 180,E1 24439.665,E2 24439.665} C_VEL
LIN {X 0,Y 520.573,Z 513.956,A -85,B 0,C 180,E1 24436.231,E2 24436.231} C_VEL
LIN {X 0,Y 520.546,Z 513.952,A -85,B 0,C 180,E1 24432.799,E2 24432.799} C_VEL
LIN {X 0,Y 520.59,Z 513.951,A -85,B 0,C 180,E1 24429.458,E2 24429.458} C_VEL
LIN {X 0,Y 520.571,Z 513.954,A -85,B 0,C 180,E1 24425.994,E2 24425.994} C_VEL
LIN {X 0,Y 520.59,Z 514.206,A -85,B 0,C 180,E1 24424.227,E2 24424.227} C_VEL
LIN {X 0,Y 527.665,Z 534.7,A -85,B 0,C 180,E1 24422.01,E2 24422.01} C_VEL
LIN {X 0,Y 526.482,Z 570.271,A -85,B 0,C 180,E1 24419.275,E2 24419.275} C_VEL
LIN {X 0,Y 525.284,Z 611.008,A -85,B 0,C 180,E1 24416.205,E2 24416.205} C_VEL
LIN {X 0,Y 525.245,Z 615.586,A -85,B 0,C 180,E1 24415.9,E2 24415.9} C_VEL
LIN {X 0,Y 526.878,Z 627.901,A -85,B 0,C 180,E1 24415.656,E2 24415.656} C_VEL
LIN {X 0,Y 525.648,Z 824.167,A -85,B 0,C 180,E1 24412.906,E2 24412.906} C_VEL
LIN {X 0,Y 525.236,Z 843.491,A -85,B 0,C 180,E1 24412.429,E2 24412.429} C_VEL
LIN {X 0,Y 524.74,Z 861.681,A -85,B 0,C 180,E1 24411.782,E2 24411.782} C_VEL
LIN {X 0,Y 524.211,Z 878.027,A -85,B 0,C 180,E1 24411.013,E2 24411.013} C_VEL
LIN {X 0,Y 523.496,Z 894.956,A -85,B 0,C 180,E1 24409.991,E2 24409.991} C_VEL
LIN {X 0,Y 522.811,Z 910.984,A -85,B 0,C 180,E1 24408.796,E2 24408.796} C_VEL
LIN {X 0,Y 522.123,Z 925.998,A -85,B 0,C 180,E1 24407.439,E2 24407.439} C_VEL
LIN {X 0,Y 521.495,Z 940.019,A -85,B 0,C 180,E1 24405.913,E2 24405.913} C_VEL
LIN {X 0,Y 520.953,Z 952.911,A -85,B 0,C 180,E1 24404.221,E2 24404.221} C_VEL
LIN {X 0,Y 520.538,Z 964.226,A -85,B 0,C 180,E1 24402.424,E2 24402.424} C_VEL
LIN {X 0,Y 520.245,Z 973.99,A -85,B 0,C 180,E1 24400.521,E2 24400.521} C_VEL
LIN {X 0,Y 520.065,Z 982.174,A -85,B 0,C 180,E1 24398.514,E2 24398.514} C_VEL
LIN {X 0,Y 519.965,Z 988.41,A -85,B 0,C 180,E1 24396.515,E2 24396.515} C_VEL
LIN {X 0,Y 519.926,Z 992.875,A -85,B 0,C 180,E1 24394.523,E2 24394.523} C_VEL
LIN {X 0,Y 519.912,Z 995.792,A -85,B 0,C 180,E1 24392.426,E2 24392.426} C_VEL
LIN {X 0,Y 519.908,Z 996.939,A -85,B 0,C 180,E1 24390.332,E2 24390.332} C_VEL
LIN {X 0,Y 519.912,Z 996.347,A -85,B 0,C 180,E1 24388.238,E2 24388.238} C_VEL
LIN {X 0,Y 519.917,Z 994.162,A -85,B 0,C 180,E1 24386.253,E2 24386.253} C_VEL
LIN {X 0,Y 519.94,Z 990.355,A -85,B 0,C 180,E1 24384.263,E2 24384.263} C_VEL
LIN {X 0,Y 520.018,Z 984.827,A -85,B 0,C 180,E1 24382.267,E2 24382.267} C_VEL
LIN {X 0,Y 520.157,Z 977.435,A -85,B 0,C 180,E1 24380.263,E2 24380.263} C_VEL
LIN {X 0,Y 520.402,Z 968.529,A -85,B 0,C 180,E1 24378.364,E2 24378.364} C_VEL
LIN {X 0,Y 520.757,Z 958.168,A -85,B 0,C 180,E1 24376.569,E2 24376.569} C_VEL
LIN {X 0,Y 521.224,Z 946.371,A -85,B 0,C 180,E1 24374.88,E2 24374.88} C_VEL
LIN {X 0,Y 521.801,Z 933.103,A -85,B 0,C 180,E1 24373.299,E2 24373.299} C_VEL
LIN {X 0,Y 522.481,Z 918.248,A -85,B 0,C 180,E1 24371.828,E2 24371.828} C_VEL
LIN {X 0,Y 523.202,Z 902.274,A -85,B 0,C 180,E1 24370.523,E2 24370.523} C_VEL
LIN {X 0,Y 523.915,Z 885.111,A -85,B 0,C 180,E1 24369.387,E2 24369.387} C_VEL
LIN {X 0,Y 524.558,Z 868.092,A -85,B 0,C 180,E1 24368.495,E2 24368.495} C_VEL
LIN {X 0,Y 525.065,Z 849.685,A -85,B 0,C 180,E1 24367.768,E2 24367.768} C_VEL
LIN {X 0,Y 525.506,Z 830.721,A -85,B 0,C 180,E1 24367.235,E2 24367.235} C_VEL
LIN {X 0,Y 525.782,Z 809.915,A -85,B 0,C 180,E1 24366.872,E2 24366.872} C_VEL
LIN {X 0,Y 526.673,Z 625.057,A -85,B 0,C 180,E1 24364.304,E2 24364.304} C_VEL
LIN {X 0,Y 525.155,Z 614.448,A -85,B 0,C 180,E1 24364.06,E2 24364.06} C_VEL
LIN {X 0,Y 526.482,Z 570.31,A -85,B 0,C 180,E1 24360.728,E2 24360.728} C_VEL
LIN {X 0,Y 527.652,Z 534.68,A -85,B 0,C 180,E1 24357.992,E2 24357.992} C_VEL
LIN {X 0,Y 520.606,Z 514.314,A -85,B 0,C 180,E1 24355.794,E2 24355.794} C_VEL
LIN {X 0,Y 520.583,Z 513.954,A -85,B 0,C 180,E1 24354.822,E2 24354.822} C_VEL
LIN {X 0,Y 520.544,Z 513.954,A -85,B 0,C 180,E1 24351.378,E2 24351.378} C_VEL
LIN {X 0,Y 520.567,Z 513.956,A -85,B 0,C 180,E1 24347.914,E2 24347.914} C_VEL
LIN {X 0,Y 520.581,Z 513.95,A -85,B 0,C 180,E1 24344.51,E2 24344.51} C_VEL
LIN {X 0,Y 520.534,Z 513.954,A -85,B 0,C 180,E1 24341.16,E2 24341.16} C_VEL
LIN {X 0,Y 520.571,Z 513.955,A -85,B 0,C 180,E1 24337.785,E2 24337.785} C_VEL
LIN {X 0,Y 520.545,Z 513.951,A -85,B 0,C 180,E1 24334.516,E2 24334.516} C_VEL
LIN {X 0,Y 520.525,Z 513.954,A -85,B 0,C 180,E1 24331.062,E2 24331.062} C_VEL
LIN {X 0,Y 520.584,Z 513.947,A -85,B 0,C 180,E1 24327.821,E2 24327.821} C_VEL
LIN {X 0,Y 520.518,Z 513.953,A -85,B 0,C 180,E1 24324.514,E2 24324.514} C_VEL
LIN {X 0,Y 520.525,Z 513.955,A -85,B 0,C 180,E1 24321.023,E2 24321.023} C_VEL
LIN {X 0,Y 520.564,Z 513.951,A -85,B 0,C 180,E1 24317.717,E2 24317.717} C_VEL
LIN {X 0,Y 520.501,Z 513.948,A -85,B 0,C 180,E1 24314.461,E2 24314.461} C_VEL
LIN {X 0,Y 520.554,Z 513.953,A -85,B 0,C 180,E1 24311.186,E2 24311.186} C_VEL
LIN {X 0,Y 520.511,Z 513.955,A -85,B 0,C 180,E1 24307.95,E2 24307.95} C_VEL
LIN {X 0,Y 520.51,Z 513.949,A -85,B 0,C 180,E1 24304.407,E2 24304.407} C_VEL
LIN {X 0,Y 520.581,Z 513.949,A -85,B 0,C 180,E1 24301.1,E2 24301.1} C_VEL
LIN {X 0,Y 520.518,Z 513.955,A -85,B 0,C 180,E1 24297.798,E2 24297.798} C_VEL
LIN {X 0,Y 520.528,Z 513.952,A -85,B 0,C 180,E1 24294.267,E2 24294.267} C_VEL
LIN {X 0,Y 520.571,Z 513.95,A -85,B 0,C 180,E1 24291.05,E2 24291.05} C_VEL
LIN {X 0,Y 520.526,Z 513.954,A -85,B 0,C 180,E1 24287.689,E2 24287.689} C_VEL
LIN {X 0,Y 520.564,Z 513.952,A -85,B 0,C 180,E1 24284.287,E2 24284.287} C_VEL
LIN {X 0,Y 520.564,Z 513.954,A -85,B 0,C 180,E1 24280.942,E2 24280.942} C_VEL
LIN {X 0,Y 520.537,Z 513.954,A -85,B 0,C 180,E1 24277.527,E2 24277.527} C_VEL
LIN {X 0,Y 520.582,Z 513.95,A -85,B 0,C 180,E1 24274.151,E2 24274.151} C_VEL
LIN {X 0,Y 520.563,Z 513.955,A -85,B 0,C 180,E1 24270.799,E2 24270.799} C_VEL
LIN {X 0,Y 520.548,Z 513.953,A -85,B 0,C 180,E1 24267.334,E2 24267.334} C_VEL
LIN {X 0,Y 520.587,Z 513.951,A -85,B 0,C 180,E1 24263.949,E2 24263.949} C_VEL
LIN {X 0,Y 520.572,Z 513.956,A -85,B 0,C 180,E1 24260.524,E2 24260.524} C_VEL
LIN {X 0,Y 520.63,Z 514.247,A -85,B 0,C 180,E1 24260.136,E2 24260.136} C_VEL
LIN {X 0,Y 522.342,Z 520.404,A -85,B 0,C 180,E1 24259.199,E2 24259.199} C_VEL
LIN {X 0,Y 522.611,Z 524.622,A -85,B 0,C 180,E1 24258.637,E2 24258.637} C_VEL
LIN {X 0,Y 521.104,Z 530.792,A -85,B 0,C 180,E1 24257.944,E2 24257.944} C_VEL
LIN {X 0,Y 517.342,Z 541.953,A -85,B 0,C 180,E1 24256.754,E2 24256.754} C_VEL
LIN {X 0,Y 516.903,Z 545.036,A -85,B 0,C 180,E1 24256.386,E2 24256.386} C_VEL
LIN {X 0,Y 515.717,Z 573.362,A -85,B 0,C 180,E1 24252.873,E2 24252.873} C_VEL
LIN {X 0,Y 514.718,Z 601.54,A -85,B 0,C 180,E1 24249.43,E2 24249.43} C_VEL
LIN {X 0,Y 513.803,Z 631.349,A -85,B 0,C 180,E1 24245.85,E2 24245.85} C_VEL
LIN {X 0,Y 513.931,Z 633.346,A -85,B 0,C 180,E1 24245.715,E2 24245.715} C_VEL
LIN {X 0,Y 515.384,Z 644.261,A -85,B 0,C 180,E1 24245.486,E2 24245.486} C_VEL
LIN {X 0,Y 514.641,Z 746.061,A -85,B 0,C 180,E1 24243.988,E2 24243.988} C_VEL
LIN {X 0,Y 514.441,Z 761.012,A -85,B 0,C 180,E1 24243.558,E2 24243.558} C_VEL
LIN {X 0,Y 514.115,Z 775.311,A -85,B 0,C 180,E1 24242.923,E2 24242.923} C_VEL
LIN {X 0,Y 513.736,Z 788.025,A -85,B 0,C 180,E1 24242.154,E2 24242.154} C_VEL
LIN {X 0,Y 513.293,Z 800.835,A -85,B 0,C 180,E1 24241.138,E2 24241.138} C_VEL
LIN {X 0,Y 512.902,Z 812.499,A -85,B 0,C 180,E1 24239.933,E2 24239.933} C_VEL
LIN {X 0,Y 512.573,Z 822.063,A -85,B 0,C 180,E1 24238.672,E2 24238.672} C_VEL
LIN {X 0,Y 512.319,Z 830.288,A -85,B 0,C 180,E1 24237.295,E2 24237.295} C_VEL
LIN {X 0,Y 512.141,Z 837.534,A -85,B 0,C 180,E1 24235.68,E2 24235.68} C_VEL
LIN {X 0,Y 512.048,Z 842.657,A -85,B 0,C 180,E1 24234.082,E2 24234.082} C_VEL
LIN {X 0,Y 512.003,Z 845.999,A -85,B 0,C 180,E1 24232.501,E2 24232.501} C_VEL
LIN {X 0,Y 511.981,Z 847.808,A -85,B 0,C 180,E1 24230.697,E2 24230.697} C_VEL
LIN {X 0,Y 511.977,Z 847.695,A -85,B 0,C 180,E1 24229.032,E2 24229.032} C_VEL
LIN {X 0,Y 511.996,Z 845.927,A -85,B 0,C 180,E1 24227.382,E2 24227.382} C_VEL
LIN {X 0,Y 512.049,Z 842.088,A -85,B 0,C 180,E1 24225.63,E2 24225.63} C_VEL
LIN {X 0,Y 512.147,Z 836.551,A -85,B 0,C 180,E1 24224,E2 24224} C_VEL
LIN {X 0,Y 512.318,Z 829.598,A -85,B 0,C 180,E1 24222.509,E2 24222.509} C_VEL
LIN {X 0,Y 512.577,Z 821.211,A -85,B 0,C 180,E1 24221.132,E2 24221.132} C_VEL
LIN {X 0,Y 512.916,Z 811.027,A -85,B 0,C 180,E1 24219.832,E2 24219.832} C_VEL
LIN {X 0,Y 513.282,Z 800.189,A -85,B 0,C 180,E1 24218.737,E2 24218.737} C_VEL
LIN {X 0,Y 513.718,Z 787.119,A -85,B 0,C 180,E1 24217.716,E2 24217.716} C_VEL
LIN {X 0,Y 514.099,Z 773.638,A -85,B 0,C 180,E1 24216.924,E2 24216.924} C_VEL
LIN {X 0,Y 514.413,Z 759.442,A -85,B 0,C 180,E1 24216.32,E2 24216.32} C_VEL
LIN {X 0,Y 514.638,Z 743.914,A -85,B 0,C 180,E1 24215.899,E2 24215.899} C_VEL
LIN {X 0,Y 515.073,Z 640.742,A -85,B 0,C 180,E1 24214.396,E2 24214.396} C_VEL
LIN {X 0,Y 513.745,Z 632.175,A -85,B 0,C 180,E1 24214.184,E2 24214.184} C_VEL
LIN {X 0,Y 514.486,Z 604.502,A -85,B 0,C 180,E1 24210.889,E2 24210.889} C_VEL
LIN {X 0,Y 515.482,Z 576.177,A -85,B 0,C 180,E1 24207.442,E2 24207.442} C_VEL
LIN {X 0,Y 516.584,Z 548.215,A -85,B 0,C 180,E1 24204,E2 24204} C_VEL
LIN {X 0,Y 517.245,Z 532.247,A -85,B 0,C 180,E1 24201.999,E2 24201.999} C_VEL
LIN {X 0,Y 512.638,Z 515.043,A -85,B 0,C 180,E1 24199.426,E2 24199.426} C_VEL
LIN {X 0,Y 512.581,Z 514.945,A -85,B 0,C 180,E1 24196.118,E2 24196.118} C_VEL
LIN {X 0,Y 512.572,Z 514.946,A -85,B 0,C 180,E1 24192.635,E2 24192.635} C_VEL
LIN {X 0,Y 512.634,Z 514.944,A -85,B 0,C 180,E1 24189.328,E2 24189.328} C_VEL
LIN {X 0,Y 512.562,Z 514.924,A -85,B 0,C 180,E1 24186.063,E2 24186.063} C_VEL
LIN {X 0,Y 512.584,Z 514.944,A -85,B 0,C 180,E1 24182.592,E2 24182.592} C_VEL
LIN {X 0,Y 512.59,Z 514.921,A -85,B 0,C 180,E1 24179.342,E2 24179.342} C_VEL
LIN {X 0,Y 512.562,Z 514.945,A -85,B 0,C 180,E1 24175.956,E2 24175.956} C_VEL
LIN {X 0,Y 512.623,Z 514.938,A -85,B 0,C 180,E1 24172.658,E2 24172.658} C_VEL
LIN {X 0,Y 512.567,Z 514.946,A -85,B 0,C 180,E1 24169.493,E2 24169.493} C_VEL
LIN {X 0,Y 512.585,Z 514.943,A -85,B 0,C 180,E1 24166.022,E2 24166.022} C_VEL
LIN {X 0,Y 512.619,Z 514.943,A -85,B 0,C 180,E1 24162.668,E2 24162.668} C_VEL
LIN {X 0,Y 512.571,Z 514.941,A -85,B 0,C 180,E1 24159.344,E2 24159.344} C_VEL
LIN {X 0,Y 512.611,Z 514.938,A -85,B 0,C 180,E1 24155.952,E2 24155.952} C_VEL
LIN {X 0,Y 512.59,Z 514.935,A -85,B 0,C 180,E1 24152.706,E2 24152.706} C_VEL
LIN {X 0,Y 512.58,Z 514.943,A -85,B 0,C 180,E1 24149.315,E2 24149.315} C_VEL
LIN {X 0,Y 512.638,Z 514.929,A -85,B 0,C 180,E1 24146.03,E2 24146.03} C_VEL
LIN {X 0,Y 512.58,Z 514.943,A -85,B 0,C 180,E1 24142.691,E2 24142.691} C_VEL
LIN {X 0,Y 512.6,Z 514.934,A -85,B 0,C 180,E1 24139.248,E2 24139.248} C_VEL
LIN {X 0,Y 512.621,Z 514.933,A -85,B 0,C 180,E1 24135.944,E2 24135.944} C_VEL
LIN {X 0,Y 512.584,Z 514.942,A -85,B 0,C 180,E1 24132.619,E2 24132.619} C_VEL
LIN {X 0,Y 512.628,Z 514.925,A -85,B 0,C 180,E1 24129.204,E2 24129.204} C_VEL
LIN {X 0,Y 512.599,Z 514.939,A -85,B 0,C 180,E1 24125.934,E2 24125.934} C_VEL
LIN {X 0,Y 512.592,Z 514.937,A -85,B 0,C 180,E1 24122.46,E2 24122.46} C_VEL
LIN {X 0,Y 512.65,Z 514.933,A -85,B 0,C 180,E1 24119.106,E2 24119.106} C_VEL
LIN {X 0,Y 512.597,Z 514.943,A -85,B 0,C 180,E1 24115.749,E2 24115.749} C_VEL
LIN {X 0,Y 512.599,Z 514.929,A -85,B 0,C 180,E1 24112.233,E2 24112.233} C_VEL
LIN {X 0,Y 512.648,Z 514.942,A -85,B 0,C 180,E1 24108.867,E2 24108.867} C_VEL
LIN {X 0,Y 512.597,Z 514.935,A -85,B 0,C 180,E1 24105.542,E2 24105.542} C_VEL
LIN {X 0,Y 512.614,Z 514.94,A -85,B 0,C 180,E1 24102.051,E2 24102.051} C_VEL
LIN {X 0,Y 512.649,Z 514.934,A -85,B 0,C 180,E1 24098.61,E2 24098.61} C_VEL
LIN {X 0,Y 512.603,Z 514.943,A -85,B 0,C 180,E1 24095.205,E2 24095.205} C_VEL
LIN {X 0,Y 512.615,Z 514.939,A -85,B 0,C 180,E1 24091.708,E2 24091.708} C_VEL
LIN {X 0,Y 512.648,Z 514.937,A -85,B 0,C 180,E1 24088.355,E2 24088.355} C_VEL
LIN {X 0,Y 512.603,Z 514.94,A -85,B 0,C 180,E1 24085.003,E2 24085.003} C_VEL
LIN {X 0,Y 512.629,Z 514.935,A -85,B 0,C 180,E1 24081.524,E2 24081.524} C_VEL
LIN {X 0,Y 512.643,Z 514.939,A -85,B 0,C 180,E1 24078.16,E2 24078.16} C_VEL
LIN {X 0,Y 512.608,Z 514.938,A -85,B 0,C 180,E1 24074.757,E2 24074.757} C_VEL
LIN {X 0,Y 512.646,Z 514.939,A -85,B 0,C 180,E1 24071.332,E2 24071.332} C_VEL
LIN {X 0,Y 512.647,Z 514.941,A -85,B 0,C 180,E1 24067.823,E2 24067.823} C_VEL
LIN {X 0,Y 512.647,Z 515.164,A -85,B 0,C 180,E1 24064.696,E2 24064.696} C_VEL
LIN {X 0,Y 520.352,Z 537.416,A -85,B 0,C 180,E1 24062.25,E2 24062.25} C_VEL
LIN {X 0,Y 519.176,Z 568.719,A -85,B 0,C 180,E1 24059.792,E2 24059.792} C_VEL
LIN {X 0,Y 517.65,Z 613.149,A -85,B 0,C 180,E1 24056.375,E2 24056.375} C_VEL
LIN {X 0,Y 517.712,Z 616.062,A -85,B 0,C 180,E1 24056.211,E2 24056.211} C_VEL
LIN {X 0,Y 519.387,Z 628.899,A -85,B 0,C 180,E1 24055.953,E2 24055.953} C_VEL
LIN {X 0,Y 518.046,Z 823.499,A -85,B 0,C 180,E1 24053.19,E2 24053.19} C_VEL
LIN {X 0,Y 517.597,Z 842.708,A -85,B 0,C 180,E1 24052.712,E2 24052.712} C_VEL
LIN {X 0,Y 517.056,Z 860.753,A -85,B 0,C 180,E1 24052.063,E2 24052.063} C_VEL
LIN {X 0,Y 516.451,Z 878.369,A -85,B 0,C 180,E1 24051.225,E2 24051.225} C_VEL
LIN {X 0,Y 515.727,Z 895.645,A -85,B 0,C 180,E1 24050.187,E2 24050.187} C_VEL
LIN {X 0,Y 515.045,Z 912.026,A -85,B 0,C 180,E1 24048.976,E2 24048.976} C_VEL
LIN {X 0,Y 514.403,Z 925.666,A -85,B 0,C 180,E1 24047.744,E2 24047.744} C_VEL
LIN {X 0,Y 513.735,Z 939.093,A -85,B 0,C 180,E1 24046.276,E2 24046.276} C_VEL
LIN {X 0,Y 513.163,Z 951.369,A -85,B 0,C 180,E1 24044.673,E2 24044.673} C_VEL
LIN {X 0,Y 512.676,Z 962.955,A -85,B 0,C 180,E1 24042.846,E2 24042.846} C_VEL
LIN {X 0,Y 512.34,Z 972.571,A -85,B 0,C 180,E1 24040.999,E2 24040.999} C_VEL
LIN {X 0,Y 512.117,Z 980.554,A -85,B 0,C 180,E1 24039.1,E2 24039.1} C_VEL
LIN {X 0,Y 511.99,Z 987.197,A -85,B 0,C 180,E1 24037.068,E2 24037.068} C_VEL
LIN {X 0,Y 511.927,Z 992.048,A -85,B 0,C 180,E1 24035.043,E2 24035.043} C_VEL
LIN {X 0,Y 511.913,Z 995.223,A -85,B 0,C 180,E1 24033.024,E2 24033.024} C_VEL
LIN {X 0,Y 511.91,Z 996.826,A -85,B 0,C 180,E1 24030.897,E2 24030.897} C_VEL
LIN {X 0,Y 511.906,Z 996.753,A -85,B 0,C 180,E1 24028.882,E2 24028.882} C_VEL
LIN {X 0,Y 511.913,Z 994.957,A -85,B 0,C 180,E1 24026.755,E2 24026.755} C_VEL
LIN {X 0,Y 511.936,Z 991.371,A -85,B 0,C 180,E1 24024.623,E2 24024.623} C_VEL
LIN {X 0,Y 512.003,Z 986.24,A -85,B 0,C 180,E1 24022.597,E2 24022.597} C_VEL
LIN {X 0,Y 512.151,Z 979.269,A -85,B 0,C 180,E1 24020.564,E2 24020.564} C_VEL
LIN {X 0,Y 512.393,Z 970.821,A -85,B 0,C 180,E1 24018.636,E2 24018.636} C_VEL
LIN {X 0,Y 512.753,Z 960.969,A -85,B 0,C 180,E1 24016.815,E2 24016.815} C_VEL
LIN {X 0,Y 513.232,Z 949.596,A -85,B 0,C 180,E1 24015.08,E2 24015.08} C_VEL
LIN {X 0,Y 513.848,Z 936.649,A -85,B 0,C 180,E1 24013.44,E2 24013.44} C_VEL
LIN {X 0,Y 514.553,Z 922.49,A -85,B 0,C 180,E1 24011.948,E2 24011.948} C_VEL
LIN {X 0,Y 515.199,Z 908.467,A -85,B 0,C 180,E1 24010.739,E2 24010.739} C_VEL
LIN {X 0,Y 515.863,Z 892.125,A -85,B 0,C 180,E1 24009.584,E2 24009.584} C_VEL
LIN {X 0,Y 516.585,Z 874.688,A -85,B 0,C 180,E1 24008.588,E2 24008.588} C_VEL
LIN {X 0,Y 517.182,Z 856.324,A -85,B 0,C 180,E1 24007.766,E2 24007.766} C_VEL
LIN {X 0,Y 517.697,Z 837.594,A -85,B 0,C 180,E1 24007.148,E2 24007.148} C_VEL
LIN {X 0,Y 518.089,Z 817.851,A -85,B 0,C 180,E1 24006.719,E2 24006.719} C_VEL
LIN {X 0,Y 519.178,Z 626.119,A -85,B 0,C 180,E1 24004.013,E2 24004.013} C_VEL
LIN {X 0,Y 517.575,Z 614.631,A -85,B 0,C 180,E1 24003.748,E2 24003.748} C_VEL
LIN {X 0,Y 519.094,Z 569.862,A -85,B 0,C 180,E1 24000.308,E2 24000.308} C_VEL
LIN {X 0,Y 520.266,Z 537.2,A -85,B 0,C 180,E1 23997.736,E2 23997.736} C_VEL
LIN {X 0,Y 513.352,Z 517.477,A -85,B 0,C 180,E1 23995.583,E2 23995.583} C_VEL
LIN {X 0,Y 512.639,Z 515.111,A -85,B 0,C 180,E1 23995.254,E2 23995.254} C_VEL
LIN {X 0,Y 512.616,Z 514.945,A -85,B 0,C 180,E1 23991.813,E2 23991.813} C_VEL
LIN {X 0,Y 512.653,Z 514.938,A -85,B 0,C 180,E1 23988.468,E2 23988.468} C_VEL
LIN {X 0,Y 512.603,Z 514.943,A -85,B 0,C 180,E1 23985.076,E2 23985.076} C_VEL
LIN {X 0,Y 512.607,Z 514.943,A -85,B 0,C 180,E1 23981.543,E2 23981.543} C_VEL
LIN {X 0,Y 512.65,Z 514.935,A -85,B 0,C 180,E1 23978.19,E2 23978.19} C_VEL
LIN {X 0,Y 512.591,Z 514.941,A -85,B 0,C 180,E1 23974.804,E2 23974.804} C_VEL
LIN {X 0,Y 512.594,Z 514.944,A -85,B 0,C 180,E1 23971.255,E2 23971.255} C_VEL
LIN {X 0,Y 512.643,Z 514.935,A -85,B 0,C 180,E1 23967.941,E2 23967.941} C_VEL
LIN {X 0,Y 512.578,Z 514.942,A -85,B 0,C 180,E1 23964.55,E2 23964.55} C_VEL
LIN {X 0,Y 512.596,Z 514.944,A -85,B 0,C 180,E1 23961.153,E2 23961.153} C_VEL
LIN {X 0,Y 512.612,Z 514.939,A -85,B 0,C 180,E1 23957.832,E2 23957.832} C_VEL
LIN {X 0,Y 512.563,Z 514.936,A -85,B 0,C 180,E1 23954.459,E2 23954.459} C_VEL
LIN {X 0,Y 512.608,Z 514.942,A -85,B 0,C 180,E1 23951.134,E2 23951.134} C_VEL
LIN {X 0,Y 512.579,Z 514.944,A -85,B 0,C 180,E1 23947.848,E2 23947.848} C_VEL
LIN {X 0,Y 512.57,Z 514.938,A -85,B 0,C 180,E1 23944.363,E2 23944.363} C_VEL
LIN {X 0,Y 512.637,Z 514.937,A -85,B 0,C 180,E1 23941.006,E2 23941.006} C_VEL
LIN {X 0,Y 512.587,Z 514.944,A -85,B 0,C 180,E1 23937.652,E2 23937.652} C_VEL
LIN {X 0,Y 512.583,Z 514.941,A -85,B 0,C 180,E1 23934.104,E2 23934.104} C_VEL
LIN {X 0,Y 512.646,Z 514.934,A -85,B 0,C 180,E1 23930.797,E2 23930.797} C_VEL
LIN {X 0,Y 512.593,Z 514.944,A -85,B 0,C 180,E1 23927.495,E2 23927.495} C_VEL
LIN {X 0,Y 512.598,Z 514.942,A -85,B 0,C 180,E1 23923.92,E2 23923.92} C_VEL
LIN {X 0,Y 512.65,Z 514.94,A -85,B 0,C 180,E1 23920.518,E2 23920.518} C_VEL
LIN {X 0,Y 512.605,Z 514.945,A -85,B 0,C 180,E1 23917.16,E2 23917.16} C_VEL
LIN {X 0,Y 512.607,Z 514.941,A -85,B 0,C 180,E1 23913.594,E2 23913.594} C_VEL
LIN {X 0,Y 512.651,Z 514.938,A -85,B 0,C 180,E1 23910.175,E2 23910.175} C_VEL
LIN {X 0,Y 512.623,Z 514.946,A -85,B 0,C 180,E1 23906.764,E2 23906.764} C_VEL
LIN {X 0,Y 512.614,Z 514.945,A -85,B 0,C 180,E1 23903.215,E2 23903.215} C_VEL
LIN {X 0,Y 512.667,Z 515.214,A -85,B 0,C 180,E1 23900.588,E2 23900.588} C_VEL
LIN {X 0,Y 517.474,Z 532.719,A -85,B 0,C 180,E1 23897.933,E2 23897.933} C_VEL
LIN {X 0,Y 516.903,Z 545.036,A -85,B 0,C 180,E1 23896.386,E2 23896.386} C_VEL
LIN {X 0,Y 515.72,Z 550.398,A -85,B 0,C 180,E1 23895.775,E2 23895.775} C_VEL
LIN {X 0,Y 509.235,Z 565.403,A -85,B 0,C 180,E1 23894.253,E2 23894.253} C_VEL
LIN {X 0,Y 508.364,Z 569.993,A -85,B 0,C 180,E1 23893.716,E2 23893.716} C_VEL
LIN {X 0,Y 507.173,Z 599.174,A -85,B 0,C 180,E1 23890.1,E2 23890.1} C_VEL
LIN {X 0,Y 506.181,Z 628.857,A -85,B 0,C 180,E1 23886.476,E2 23886.476} C_VEL
LIN {X 0,Y 506.143,Z 632.522,A -85,B 0,C 180,E1 23886.08,E2 23886.08} C_VEL
LIN {X 0,Y 507.92,Z 644.628,A -85,B 0,C 180,E1 23885.806,E2 23885.806} C_VEL
LIN {X 0,Y 507.08,Z 746.785,A -85,B 0,C 180,E1 23884.272,E2 23884.272} C_VEL
LIN {X 0,Y 506.86,Z 761.989,A -85,B 0,C 180,E1 23883.825,E2 23883.825} C_VEL
LIN {X 0,Y 506.488,Z 776.928,A -85,B 0,C 180,E1 23883.145,E2 23883.145} C_VEL
LIN {X 0,Y 506.041,Z 790.37,A -85,B 0,C 180,E1 23882.296,E2 23882.296} C_VEL
LIN {X 0,Y 505.584,Z 802.359,A -85,B 0,C 180,E1 23881.313,E2 23881.313} C_VEL
LIN {X 0,Y 505.141,Z 814.287,A -85,B 0,C 180,E1 23880.047,E2 23880.047} C_VEL
LIN {X 0,Y 504.741,Z 824.509,A -85,B 0,C 180,E1 23878.641,E2 23878.641} C_VEL
LIN {X 0,Y 504.458,Z 832.398,A -85,B 0,C 180,E1 23877.244,E2 23877.244} C_VEL
LIN {X 0,Y 504.276,Z 838.94,A -85,B 0,C 180,E1 23875.732,E2 23875.732} C_VEL
LIN {X 0,Y 504.16,Z 843.977,A -85,B 0,C 180,E1 23874.11,E2 23874.11} C_VEL
LIN {X 0,Y 504.096,Z 847.347,A -85,B 0,C 180,E1 23872.436,E2 23872.436} C_VEL
LIN {X 0,Y 504.071,Z 849.013,A -85,B 0,C 180,E1 23870.672,E2 23870.672} C_VEL
LIN {X 0,Y 504.067,Z 848.794,A -85,B 0,C 180,E1 23868.884,E2 23868.884} C_VEL
LIN {X 0,Y 504.093,Z 846.835,A -85,B 0,C 180,E1 23867.187,E2 23867.187} C_VEL
LIN {X 0,Y 504.166,Z 842.986,A -85,B 0,C 180,E1 23865.455,E2 23865.455} C_VEL
LIN {X 0,Y 504.301,Z 836.977,A -85,B 0,C 180,E1 23863.709,E2 23863.709} C_VEL
LIN {X 0,Y 504.506,Z 830.013,A -85,B 0,C 180,E1 23862.241,E2 23862.241} C_VEL
LIN {X 0,Y 504.816,Z 821.458,A -85,B 0,C 180,E1 23860.843,E2 23860.843} C_VEL
LIN {X 0,Y 505.232,Z 810.431,A -85,B 0,C 180,E1 23859.452,E2 23859.452} C_VEL
LIN {X 0,Y 505.658,Z 798.595,A -85,B 0,C 180,E1 23858.297,E2 23858.297} C_VEL
LIN {X 0,Y 506.112,Z 786.365,A -85,B 0,C 180,E1 23857.368,E2 23857.368} C_VEL
LIN {X 0,Y 506.526,Z 772.563,A -85,B 0,C 180,E1 23856.572,E2 23856.572} C_VEL
LIN {X 0,Y 506.859,Z 757.748,A -85,B 0,C 180,E1 23855.971,E2 23855.971} C_VEL
LIN {X 0,Y 507.063,Z 742.949,A -85,B 0,C 180,E1 23855.592,E2 23855.592} C_VEL
LIN {X 0,Y 507.581,Z 641.726,A -85,B 0,C 180,E1 23854.097,E2 23854.097} C_VEL
LIN {X 0,Y 506.022,Z 632.004,A -85,B 0,C 180,E1 23853.85,E2 23853.85} C_VEL
LIN {X 0,Y 506.938,Z 602.374,A -85,B 0,C 180,E1 23850.272,E2 23850.272} C_VEL
LIN {X 0,Y 508.042,Z 573.64,A -85,B 0,C 180,E1 23846.727,E2 23846.727} C_VEL
LIN {X 0,Y 509.306,Z 544.827,A -85,B 0,C 180,E1 23843.121,E2 23843.121} C_VEL
LIN {X 0,Y 509.615,Z 534.229,A -85,B 0,C 180,E1 23841.765,E2 23841.765} C_VEL
LIN {X 0,Y 504.661,Z 516.049,A -85,B 0,C 180,E1 23839.006,E2 23839.006} C_VEL
LIN {X 0,Y 504.685,Z 515.934,A -85,B 0,C 180,E1 23835.648,E2 23835.648} C_VEL
LIN {X 0,Y 504.63,Z 515.934,A -85,B 0,C 180,E1 23832.234,E2 23832.234} C_VEL
LIN {X 0,Y 504.645,Z 515.935,A -85,B 0,C 180,E1 23828.742,E2 23828.742} C_VEL
LIN {X 0,Y 504.656,Z 515.913,A -85,B 0,C 180,E1 23825.539,E2 23825.539} C_VEL
LIN {X 0,Y 504.624,Z 515.933,A -85,B 0,C 180,E1 23822.093,E2 23822.093} C_VEL
LIN {X 0,Y 504.667,Z 515.911,A -85,B 0,C 180,E1 23818.731,E2 23818.731} C_VEL
LIN {X 0,Y 504.635,Z 515.934,A -85,B 0,C 180,E1 23815.484,E2 23815.484} C_VEL
LIN {X 0,Y 504.629,Z 515.931,A -85,B 0,C 180,E1 23811.962,E2 23811.962} C_VEL
LIN {X 0,Y 504.702,Z 515.926,A -85,B 0,C 180,E1 23808.663,E2 23808.663} C_VEL
LIN {X 0,Y 504.634,Z 515.932,A -85,B 0,C 180,E1 23805.304,E2 23805.304} C_VEL
LIN {X 0,Y 504.634,Z 515.923,A -85,B 0,C 180,E1 23801.675,E2 23801.675} C_VEL
LIN {X 0,Y 504.703,Z 515.933,A -85,B 0,C 180,E1 23798.322,E2 23798.322} C_VEL
LIN {X 0,Y 504.641,Z 515.927,A -85,B 0,C 180,E1 23794.893,E2 23794.893} C_VEL
LIN {X 0,Y 504.641,Z 515.932,A -85,B 0,C 180,E1 23791.361,E2 23791.361} C_VEL
LIN {X 0,Y 504.706,Z 515.923,A -85,B 0,C 180,E1 23788.003,E2 23788.003} C_VEL
LIN {X 0,Y 504.648,Z 515.923,A -85,B 0,C 180,E1 23784.583,E2 23784.583} C_VEL
LIN {X 0,Y 504.644,Z 515.931,A -85,B 0,C 180,E1 23781.016,E2 23781.016} C_VEL
LIN {X 0,Y 504.702,Z 515.914,A -85,B 0,C 180,E1 23777.645,E2 23777.645} C_VEL
LIN {X 0,Y 504.65,Z 515.93,A -85,B 0,C 180,E1 23774.339,E2 23774.339} C_VEL
LIN {X 0,Y 504.649,Z 515.925,A -85,B 0,C 180,E1 23770.734,E2 23770.734} C_VEL
LIN {X 0,Y 504.713,Z 515.919,A -85,B 0,C 180,E1 23767.399,E2 23767.399} C_VEL
LIN {X 0,Y 504.656,Z 515.932,A -85,B 0,C 180,E1 23763.977,E2 23763.977} C_VEL
LIN {X 0,Y 504.654,Z 515.913,A -85,B 0,C 180,E1 23760.454,E2 23760.454} C_VEL
LIN {X 0,Y 504.707,Z 515.931,A -85,B 0,C 180,E1 23757.048,E2 23757.048} C_VEL
LIN {X 0,Y 504.662,Z 515.928,A -85,B 0,C 180,E1 23753.63,E2 23753.63} C_VEL
LIN {X 0,Y 504.658,Z 515.928,A -85,B 0,C 180,E1 23750.075,E2 23750.075} C_VEL
LIN {X 0,Y 504.711,Z 515.921,A -85,B 0,C 180,E1 23746.715,E2 23746.715} C_VEL
LIN {X 0,Y 504.667,Z 515.928,A -85,B 0,C 180,E1 23743.305,E2 23743.305} C_VEL
LIN {X 0,Y 504.666,Z 515.924,A -85,B 0,C 180,E1 23739.835,E2 23739.835} C_VEL
LIN {X 0,Y 504.713,Z 515.929,A -85,B 0,C 180,E1 23736.411,E2 23736.411} C_VEL
LIN {X 0,Y 504.67,Z 515.924,A -85,B 0,C 180,E1 23733.019,E2 23733.019} C_VEL
LIN {X 0,Y 504.669,Z 515.926,A -85,B 0,C 180,E1 23729.517,E2 23729.517} C_VEL
LIN {X 0,Y 504.711,Z 515.927,A -85,B 0,C 180,E1 23726.1,E2 23726.1} C_VEL
LIN {X 0,Y 504.68,Z 515.933,A -85,B 0,C 180,E1 23722.599,E2 23722.599} C_VEL
LIN {X 0,Y 504.673,Z 515.93,A -85,B 0,C 180,E1 23719.172,E2 23719.172} C_VEL
LIN {X 0,Y 504.71,Z 515.924,A -85,B 0,C 180,E1 23715.653,E2 23715.653} C_VEL
LIN {X 0,Y 504.691,Z 515.93,A -85,B 0,C 180,E1 23712.188,E2 23712.188} C_VEL
LIN {X 0,Y 504.672,Z 515.932,A -85,B 0,C 180,E1 23708.685,E2 23708.685} C_VEL
LIN {X 0,Y 504.732,Z 516.128,A -85,B 0,C 180,E1 23705.181,E2 23705.181} C_VEL
LIN {X 0,Y 507.665,Z 524.546,A -85,B 0,C 180,E1 23704.188,E2 23704.188} C_VEL
LIN {X 0,Y 513.079,Z 540.533,A -85,B 0,C 180,E1 23702.456,E2 23702.456} C_VEL
LIN {X 0,Y 511.4,Z 579.037,A -85,B 0,C 180,E1 23699.388,E2 23699.388} C_VEL
LIN {X 0,Y 510.063,Z 615.304,A -85,B 0,C 180,E1 23696.564,E2 23696.564} C_VEL
LIN {X 0,Y 511.909,Z 629.921,A -85,B 0,C 180,E1 23696.258,E2 23696.258} C_VEL
LIN {X 0,Y 510.451,Z 822.986,A -85,B 0,C 180,E1 23693.479,E2 23693.479} C_VEL
LIN {X 0,Y 509.963,Z 842.077,A -85,B 0,C 180,E1 23692.998,E2 23692.998} C_VEL
LIN {X 0,Y 509.362,Z 860.488,A -85,B 0,C 180,E1 23692.323,E2 23692.323} C_VEL
LIN {X 0,Y 508.686,Z 878.506,A -85,B 0,C 180,E1 23691.444,E2 23691.444} C_VEL
LIN {X 0,Y 507.909,Z 895.589,A -85,B 0,C 180,E1 23690.391,E2 23690.391} C_VEL
LIN {X 0,Y 507.177,Z 911.817,A -85,B 0,C 180,E1 23689.162,E2 23689.162} C_VEL
LIN {X 0,Y 506.404,Z 927.7,A -85,B 0,C 180,E1 23687.702,E2 23687.702} C_VEL
LIN {X 0,Y 505.745,Z 941.426,A -85,B 0,C 180,E1 23686.186,E2 23686.186} C_VEL
LIN {X 0,Y 505.191,Z 953.537,A -85,B 0,C 180,E1 23684.576,E2 23684.576} C_VEL
LIN {X 0,Y 504.682,Z 964.859,A -85,B 0,C 180,E1 23682.704,E2 23682.704} C_VEL
LIN {X 0,Y 504.323,Z 974.504,A -85,B 0,C 180,E1 23680.741,E2 23680.741} C_VEL
LIN {X 0,Y 504.099,Z 982.173,A -85,B 0,C 180,E1 23678.786,E2 23678.786} C_VEL
LIN {X 0,Y 503.98,Z 988.41,A -85,B 0,C 180,E1 23676.723,E2 23676.723} C_VEL
LIN {X 0,Y 503.929,Z 992.874,A -85,B 0,C 180,E1 23674.667,E2 23674.667} C_VEL
LIN {X 0,Y 503.911,Z 995.791,A -85,B 0,C 180,E1 23672.503,E2 23672.503} C_VEL
LIN {X 0,Y 503.908,Z 996.939,A -85,B 0,C 180,E1 23670.342,E2 23670.342} C_VEL
LIN {X 0,Y 503.912,Z 996.414,A -85,B 0,C 180,E1 23668.296,E2 23668.296} C_VEL
LIN {X 0,Y 503.921,Z 994.161,A -85,B 0,C 180,E1 23666.134,E2 23666.134} C_VEL
LIN {X 0,Y 503.95,Z 990.354,A -85,B 0,C 180,E1 23664.08,E2 23664.08} C_VEL
LIN {X 0,Y 504.042,Z 984.827,A -85,B 0,C 180,E1 23662.02,E2 23662.02} C_VEL
LIN {X 0,Y 504.234,Z 977.435,A -85,B 0,C 180,E1 23659.953,E2 23659.953} C_VEL
LIN {X 0,Y 504.537,Z 968.528,A -85,B 0,C 180,E1 23657.992,E2 23657.992} C_VEL
LIN {X 0,Y 504.976,Z 958.166,A -85,B 0,C 180,E1 23656.141,E2 23656.141} C_VEL
LIN {X 0,Y 505.452,Z 947.899,A -85,B 0,C 180,E1 23654.632,E2 23654.632} C_VEL
LIN {X 0,Y 506.084,Z 934.191,A -85,B 0,C 180,E1 23652.985,E2 23652.985} C_VEL
LIN {X 0,Y 506.819,Z 919.161,A -85,B 0,C 180,E1 23651.484,E2 23651.484} C_VEL
LIN {X 0,Y 507.545,Z 903.65,A -85,B 0,C 180,E1 23650.197,E2 23650.197} C_VEL
LIN {X 0,Y 508.259,Z 887.383,A -85,B 0,C 180,E1 23649.084,E2 23649.084} C_VEL
LIN {X 0,Y 508.98,Z 870.471,A -85,B 0,C 180,E1 23648.148,E2 23648.148} C_VEL
LIN {X 0,Y 509.617,Z 852.136,A -85,B 0,C 180,E1 23647.357,E2 23647.357} C_VEL
LIN {X 0,Y 510.169,Z 833.536,A -85,B 0,C 180,E1 23646.774,E2 23646.774} C_VEL
LIN {X 0,Y 510.536,Z 814.399,A -85,B 0,C 180,E1 23646.385,E2 23646.385} C_VEL
LIN {X 0,Y 511.674,Z 627.05,A -85,B 0,C 180,E1 23643.71,E2 23643.71} C_VEL
LIN {X 0,Y 510.018,Z 615.305,A -85,B 0,C 180,E1 23643.454,E2 23643.454} C_VEL
LIN {X 0,Y 511.662,Z 570.373,A -85,B 0,C 180,E1 23639.961,E2 23639.961} C_VEL
LIN {X 0,Y 512.985,Z 540.028,A -85,B 0,C 180,E1 23637.509,E2 23637.509} C_VEL
LIN {X 0,Y 506.153,Z 520.514,A -85,B 0,C 180,E1 23635.33,E2 23635.33} C_VEL
LIN {X 0,Y 504.733,Z 516.122,A -85,B 0,C 180,E1 23634.768,E2 23634.768} C_VEL
LIN {X 0,Y 504.669,Z 515.931,A -85,B 0,C 180,E1 23631.315,E2 23631.315} C_VEL
LIN {X 0,Y 504.682,Z 515.933,A -85,B 0,C 180,E1 23627.813,E2 23627.813} C_VEL
LIN {X 0,Y 504.71,Z 515.926,A -85,B 0,C 180,E1 23624.351,E2 23624.351} C_VEL
LIN {X 0,Y 504.659,Z 515.931,A -85,B 0,C 180,E1 23620.98,E2 23620.98} C_VEL
LIN {X 0,Y 504.662,Z 515.934,A -85,B 0,C 180,E1 23617.403,E2 23617.403} C_VEL
LIN {X 0,Y 504.707,Z 515.93,A -85,B 0,C 180,E1 23613.963,E2 23613.963} C_VEL
LIN {X 0,Y 504.653,Z 515.931,A -85,B 0,C 180,E1 23610.61,E2 23610.61} C_VEL
LIN {X 0,Y 504.65,Z 515.933,A -85,B 0,C 180,E1 23607.11,E2 23607.11} C_VEL
LIN {X 0,Y 504.704,Z 515.923,A -85,B 0,C 180,E1 23603.713,E2 23603.713} C_VEL
LIN {X 0,Y 504.637,Z 515.933,A -85,B 0,C 180,E1 23600.409,E2 23600.409} C_VEL
LIN {X 0,Y 504.637,Z 515.935,A -85,B 0,C 180,E1 23596.814,E2 23596.814} C_VEL
LIN {X 0,Y 504.692,Z 515.925,A -85,B 0,C 180,E1 23593.438,E2 23593.438} C_VEL
LIN {X 0,Y 504.63,Z 515.93,A -85,B 0,C 180,E1 23590.041,E2 23590.041} C_VEL
LIN {X 0,Y 504.631,Z 515.934,A -85,B 0,C 180,E1 23586.484,E2 23586.484} C_VEL
LIN {X 0,Y 504.693,Z 515.929,A -85,B 0,C 180,E1 23583.18,E2 23583.18} C_VEL
LIN {X 0,Y 504.636,Z 515.927,A -85,B 0,C 180,E1 23579.886,E2 23579.886} C_VEL
LIN {X 0,Y 504.651,Z 515.93,A -85,B 0,C 180,E1 23576.365,E2 23576.365} C_VEL
LIN {X 0,Y 504.71,Z 515.932,A -85,B 0,C 180,E1 23572.931,E2 23572.931} C_VEL
LIN {X 0,Y 504.654,Z 515.929,A -85,B 0,C 180,E1 23569.497,E2 23569.497} C_VEL
LIN {X 0,Y 504.654,Z 515.927,A -85,B 0,C 180,E1 23565.895,E2 23565.895} C_VEL
LIN {X 0,Y 504.708,Z 515.924,A -85,B 0,C 180,E1 23562.475,E2 23562.475} C_VEL
LIN {X 0,Y 504.68,Z 515.929,A -85,B 0,C 180,E1 23558.986,E2 23558.986} C_VEL
LIN {X 0,Y 504.662,Z 515.926,A -85,B 0,C 180,E1 23555.538,E2 23555.538} C_VEL
LIN {X 0,Y 504.71,Z 515.929,A -85,B 0,C 180,E1 23552.061,E2 23552.061} C_VEL
LIN {X 0,Y 504.698,Z 515.932,A -85,B 0,C 180,E1 23548.598,E2 23548.598} C_VEL
LIN {X 0,Y 504.671,Z 515.934,A -85,B 0,C 180,E1 23545.097,E2 23545.097} C_VEL
LIN {X 0,Y 504.705,Z 515.933,A -85,B 0,C 180,E1 23541.666,E2 23541.666} C_VEL
LIN {X 0,Y 504.717,Z 516.224,A -85,B 0,C 180,E1 23541.061,E2 23541.061} C_VEL
LIN {X 0,Y 509.585,Z 533.456,A -85,B 0,C 180,E1 23538.372,E2 23538.372} C_VEL
LIN {X 0,Y 509.963,Z 536.184,A -85,B 0,C 180,E1 23537.987,E2 23537.987} C_VEL
LIN {X 0,Y 508.607,Z 564.004,A -85,B 0,C 180,E1 23534.47,E2 23534.47} C_VEL
LIN {X 0,Y 508.364,Z 569.993,A -85,B 0,C 180,E1 23533.716,E2 23533.716} C_VEL
LIN {X 0,Y 507.235,Z 575.359,A -85,B 0,C 180,E1 23533.097,E2 23533.097} C_VEL
LIN {X 0,Y 500.439,Z 591.159,A -85,B 0,C 180,E1 23531.466,E2 23531.466} C_VEL
LIN {X 0,Y 499.753,Z 595.024,A -85,B 0,C 180,E1 23531.013,E2 23531.013} C_VEL
LIN {X 0,Y 498.683,Z 622.931,A -85,B 0,C 180,E1 23527.549,E2 23527.549} C_VEL
LIN {X 0,Y 498.445,Z 632.143,A -85,B 0,C 180,E1 23526.448,E2 23526.448} C_VEL
LIN {X 0,Y 500.471,Z 645.338,A -85,B 0,C 180,E1 23526.131,E2 23526.131} C_VEL
LIN {X 0,Y 499.539,Z 747.241,A -85,B 0,C 180,E1 23524.571,E2 23524.571} C_VEL
LIN {X 0,Y 499.309,Z 761.998,A -85,B 0,C 180,E1 23524.137,E2 23524.137} C_VEL
LIN {X 0,Y 498.93,Z 776.469,A -85,B 0,C 180,E1 23523.483,E2 23523.483} C_VEL
LIN {X 0,Y 498.462,Z 789.891,A -85,B 0,C 180,E1 23522.65,E2 23522.65} C_VEL
LIN {X 0,Y 497.93,Z 802.73,A -85,B 0,C 180,E1 23521.603,E2 23521.603} C_VEL
LIN {X 0,Y 497.442,Z 814.418,A -85,B 0,C 180,E1 23520.361,E2 23520.361} C_VEL
LIN {X 0,Y 497.047,Z 823.617,A -85,B 0,C 180,E1 23519.126,E2 23519.126} C_VEL
LIN {X 0,Y 496.675,Z 832.637,A -85,B 0,C 180,E1 23517.578,E2 23517.578} C_VEL
LIN {X 0,Y 496.423,Z 839.859,A -85,B 0,C 180,E1 23515.913,E2 23515.913} C_VEL
LIN {X 0,Y 496.276,Z 844.977,A -85,B 0,C 180,E1 23514.264,E2 23514.264} C_VEL
LIN {X 0,Y 496.195,Z 848.504,A -85,B 0,C 180,E1 23512.507,E2 23512.507} C_VEL
LIN {X 0,Y 496.16,Z 850.217,A -85,B 0,C 180,E1 23510.647,E2 23510.647} C_VEL
LIN {X 0,Y 496.155,Z 849.934,A -85,B 0,C 180,E1 23508.807,E2 23508.807} C_VEL
LIN {X 0,Y 496.191,Z 847.952,A -85,B 0,C 180,E1 23507.107,E2 23507.107} C_VEL
LIN {X 0,Y 496.275,Z 844.269,A -85,B 0,C 180,E1 23505.42,E2 23505.42} C_VEL
LIN {X 0,Y 496.419,Z 838.708,A -85,B 0,C 180,E1 23503.746,E2 23503.746} C_VEL
LIN {X 0,Y 496.659,Z 831.691,A -85,B 0,C 180,E1 23502.201,E2 23502.201} C_VEL
LIN {X 0,Y 496.995,Z 823.279,A -85,B 0,C 180,E1 23500.781,E2 23500.781} C_VEL
LIN {X 0,Y 497.402,Z 813.476,A -85,B 0,C 180,E1 23499.485,E2 23499.485} C_VEL
LIN {X 0,Y 497.866,Z 802.272,A -85,B 0,C 180,E1 23498.312,E2 23498.312} C_VEL
LIN {X 0,Y 498.383,Z 789.253,A -85,B 0,C 180,E1 23497.259,E2 23497.259} C_VEL
LIN {X 0,Y 498.831,Z 775.943,A -85,B 0,C 180,E1 23496.443,E2 23496.443} C_VEL
LIN {X 0,Y 499.212,Z 761.446,A -85,B 0,C 180,E1 23495.796,E2 23495.796} C_VEL
LIN {X 0,Y 499.474,Z 745.567,A -85,B 0,C 180,E1 23495.343,E2 23495.343} C_VEL
LIN {X 0,Y 500.08,Z 642.55,A -85,B 0,C 180,E1 23493.785,E2 23493.785} C_VEL
LIN {X 0,Y 498.336,Z 632.255,A -85,B 0,C 180,E1 23493.535,E2 23493.535} C_VEL
LIN {X 0,Y 499.243,Z 604.103,A -85,B 0,C 180,E1 23490.113,E2 23490.113} C_VEL
LIN {X 0,Y 500.464,Z 574.745,A -85,B 0,C 180,E1 23486.448,E2 23486.448} C_VEL
LIN {X 0,Y 501.842,Z 545.904,A -85,B 0,C 180,E1 23482.788,E2 23482.788} C_VEL
LIN {X 0,Y 502.168,Z 536.959,A -85,B 0,C 180,E1 23481.642,E2 23481.642} C_VEL
LIN {X 0,Y 497.129,Z 518.71,A -85,B 0,C 180,E1 23478.867,E2 23478.867} C_VEL
LIN {X 0,Y 496.709,Z 517.05,A -85,B 0,C 180,E1 23478.569,E2 23478.569} C_VEL
LIN {X 0,Y 496.732,Z 516.922,A -85,B 0,C 180,E1 23475.189,E2 23475.189} C_VEL
LIN {X 0,Y 496.713,Z 516.923,A -85,B 0,C 180,E1 23471.82,E2 23471.82} C_VEL
LIN {X 0,Y 496.689,Z 516.924,A -85,B 0,C 180,E1 23468.384,E2 23468.384} C_VEL
LIN {X 0,Y 496.739,Z 516.908,A -85,B 0,C 180,E1 23464.996,E2 23464.996} C_VEL
LIN {X 0,Y 496.701,Z 516.922,A -85,B 0,C 180,E1 23461.605,E2 23461.605} C_VEL
LIN {X 0,Y 496.686,Z 516.911,A -85,B 0,C 180,E1 23458.159,E2 23458.159} C_VEL
LIN {X 0,Y 496.75,Z 516.922,A -85,B 0,C 180,E1 23454.806,E2 23454.806} C_VEL
LIN {X 0,Y 496.699,Z 516.92,A -85,B 0,C 180,E1 23451.357,E2 23451.357} C_VEL
LIN {X 0,Y 496.69,Z 516.914,A -85,B 0,C 180,E1 23447.8,E2 23447.8} C_VEL
LIN {X 0,Y 496.748,Z 516.922,A -85,B 0,C 180,E1 23444.397,E2 23444.397} C_VEL
LIN {X 0,Y 496.704,Z 516.912,A -85,B 0,C 180,E1 23440.99,E2 23440.99} C_VEL
LIN {X 0,Y 496.697,Z 516.922,A -85,B 0,C 180,E1 23437.525,E2 23437.525} C_VEL
LIN {X 0,Y 496.757,Z 516.906,A -85,B 0,C 180,E1 23434.164,E2 23434.164} C_VEL
LIN {X 0,Y 496.707,Z 516.922,A -85,B 0,C 180,E1 23430.741,E2 23430.741} C_VEL
LIN {X 0,Y 496.701,Z 516.911,A -85,B 0,C 180,E1 23427.165,E2 23427.165} C_VEL
LIN {X 0,Y 496.756,Z 516.919,A -85,B 0,C 180,E1 23423.738,E2 23423.738} C_VEL
LIN {X 0,Y 496.716,Z 516.921,A -85,B 0,C 180,E1 23420.38,E2 23420.38} C_VEL
LIN {X 0,Y 496.704,Z 516.907,A -85,B 0,C 180,E1 23416.85,E2 23416.85} C_VEL
LIN {X 0,Y 496.766,Z 516.919,A -85,B 0,C 180,E1 23413.502,E2 23413.502} C_VEL
LIN {X 0,Y 496.718,Z 516.915,A -85,B 0,C 180,E1 23410.086,E2 23410.086} C_VEL
LIN {X 0,Y 496.712,Z 516.915,A -85,B 0,C 180,E1 23406.589,E2 23406.589} C_VEL
LIN {X 0,Y 496.768,Z 516.914,A -85,B 0,C 180,E1 23403.231,E2 23403.231} C_VEL
LIN {X 0,Y 496.72,Z 516.903,A -85,B 0,C 180,E1 23399.77,E2 23399.77} C_VEL
LIN {X 0,Y 496.715,Z 516.92,A -85,B 0,C 180,E1 23396.191,E2 23396.191} C_VEL
LIN {X 0,Y 496.761,Z 516.902,A -85,B 0,C 180,E1 23392.715,E2 23392.715} C_VEL
LIN {X 0,Y 496.747,Z 516.92,A -85,B 0,C 180,E1 23389.211,E2 23389.211} C_VEL
LIN {X 0,Y 496.718,Z 516.911,A -85,B 0,C 180,E1 23385.784,E2 23385.784} C_VEL
LIN {X 0,Y 496.757,Z 516.917,A -85,B 0,C 180,E1 23382.306,E2 23382.306} C_VEL
LIN {X 0,Y 496.761,Z 516.91,A -85,B 0,C 180,E1 23378.759,E2 23378.759} C_VEL
LIN {X 0,Y 496.722,Z 516.92,A -85,B 0,C 180,E1 23375.375,E2 23375.375} C_VEL
LIN {X 0,Y 496.745,Z 516.917,A -85,B 0,C 180,E1 23371.831,E2 23371.831} C_VEL
LIN {X 0,Y 496.77,Z 516.913,A -85,B 0,C 180,E1 23368.357,E2 23368.357} C_VEL
LIN {X 0,Y 496.73,Z 516.919,A -85,B 0,C 180,E1 23364.853,E2 23364.853} C_VEL
LIN {X 0,Y 496.736,Z 516.914,A -85,B 0,C 180,E1 23361.245,E2 23361.245} C_VEL
LIN {X 0,Y 496.77,Z 516.915,A -85,B 0,C 180,E1 23357.786,E2 23357.786} C_VEL
LIN {X 0,Y 496.752,Z 516.919,A -85,B 0,C 180,E1 23354.229,E2 23354.229} C_VEL
LIN {X 0,Y 496.732,Z 516.921,A -85,B 0,C 180,E1 23350.703,E2 23350.703} C_VEL
LIN {X 0,Y 496.767,Z 516.92,A -85,B 0,C 180,E1 23347.287,E2 23347.287} C_VEL
LIN {X 0,Y 496.802,Z 517.146,A -85,B 0,C 180,E1 23345.667,E2 23345.667} C_VEL
LIN {X 0,Y 504.681,Z 539.804,A -85,B 0,C 180,E1 23343.067,E2 23343.067} C_VEL
LIN {X 0,Y 505.743,Z 543.662,A -85,B 0,C 180,E1 23342.663,E2 23342.663} C_VEL
LIN {X 0,Y 503.646,Z 587.502,A -85,B 0,C 180,E1 23339.102,E2 23339.102} C_VEL
LIN {X 0,Y 502.535,Z 615.632,A -85,B 0,C 180,E1 23336.893,E2 23336.893} C_VEL
LIN {X 0,Y 504.444,Z 630.942,A -85,B 0,C 180,E1 23336.572,E2 23336.572} C_VEL
LIN {X 0,Y 502.873,Z 822.265,A -85,B 0,C 180,E1 23333.781,E2 23333.781} C_VEL
LIN {X 0,Y 502.342,Z 841.344,A -85,B 0,C 180,E1 23333.294,E2 23333.294} C_VEL
LIN {X 0,Y 501.708,Z 859.535,A -85,B 0,C 180,E1 23332.62,E2 23332.62} C_VEL
LIN {X 0,Y 501.029,Z 876.552,A -85,B 0,C 180,E1 23331.788,E2 23331.788} C_VEL
LIN {X 0,Y 500.176,Z 893.843,A -85,B 0,C 180,E1 23330.721,E2 23330.721} C_VEL
LIN {X 0,Y 499.382,Z 910.218,A -85,B 0,C 180,E1 23329.473,E2 23329.473} C_VEL
LIN {X 0,Y 498.585,Z 925.625,A -85,B 0,C 180,E1 23328.049,E2 23328.049} C_VEL
LIN {X 0,Y 497.847,Z 940.009,A -85,B 0,C 180,E1 23326.45,E2 23326.45} C_VEL
LIN {X 0,Y 497.22,Z 953.255,A -85,B 0,C 180,E1 23324.677,E2 23324.677} C_VEL
LIN {X 0,Y 496.707,Z 964.887,A -85,B 0,C 180,E1 23322.793,E2 23322.793} C_VEL
LIN {X 0,Y 496.365,Z 974.366,A -85,B 0,C 180,E1 23320.915,E2 23320.915} C_VEL
LIN {X 0,Y 496.133,Z 981.768,A -85,B 0,C 180,E1 23319.045,E2 23319.045} C_VEL
LIN {X 0,Y 495.994,Z 988.106,A -85,B 0,C 180,E1 23316.948,E2 23316.948} C_VEL
LIN {X 0,Y 495.93,Z 992.874,A -85,B 0,C 180,E1 23314.743,E2 23314.743} C_VEL
LIN {X 0,Y 495.911,Z 995.677,A -85,B 0,C 180,E1 23312.659,E2 23312.659} C_VEL
LIN {X 0,Y 495.908,Z 996.916,A -85,B 0,C 180,E1 23310.463,E2 23310.463} C_VEL
LIN {X 0,Y 495.912,Z 996.413,A -85,B 0,C 180,E1 23308.269,E2 23308.269} C_VEL
LIN {X 0,Y 495.922,Z 994.16,A -85,B 0,C 180,E1 23306.071,E2 23306.071} C_VEL
LIN {X 0,Y 495.956,Z 990.354,A -85,B 0,C 180,E1 23303.984,E2 23303.984} C_VEL
LIN {X 0,Y 496.057,Z 984.827,A -85,B 0,C 180,E1 23301.891,E2 23301.891} C_VEL
LIN {X 0,Y 496.254,Z 977.857,A -85,B 0,C 180,E1 23299.907,E2 23299.907} C_VEL
LIN {X 0,Y 496.536,Z 969.291,A -85,B 0,C 180,E1 23298.032,E2 23298.032} C_VEL
LIN {X 0,Y 496.972,Z 958.619,A -85,B 0,C 180,E1 23296.151,E2 23296.151} C_VEL
LIN {X 0,Y 497.534,Z 946.472,A -85,B 0,C 180,E1 23294.381,E2 23294.381} C_VEL
LIN {X 0,Y 498.201,Z 932.814,A -85,B 0,C 180,E1 23292.724,E2 23292.724} C_VEL
LIN {X 0,Y 498.961,Z 918.171,A -85,B 0,C 180,E1 23291.242,E2 23291.242} C_VEL
LIN {X 0,Y 499.735,Z 902.654,A -85,B 0,C 180,E1 23289.935,E2 23289.935} C_VEL
LIN {X 0,Y 500.515,Z 886.367,A -85,B 0,C 180,E1 23288.806,E2 23288.806} C_VEL
LIN {X 0,Y 501.284,Z 869.407,A -85,B 0,C 180,E1 23287.857,E2 23287.857} C_VEL
LIN {X 0,Y 501.946,Z 851.678,A -85,B 0,C 180,E1 23287.081,E2 23287.081} C_VEL
LIN {X 0,Y 502.546,Z 833.167,A -85,B 0,C 180,E1 23286.49,E2 23286.49} C_VEL
LIN {X 0,Y 502.945,Z 814.126,A -85,B 0,C 180,E1 23286.095,E2 23286.095} C_VEL
LIN {X 0,Y 504.203,Z 628.103,A -85,B 0,C 180,E1 23283.401,E2 23283.401} C_VEL
LIN {X 0,Y 502.464,Z 615.394,A -85,B 0,C 180,E1 23283.119,E2 23283.119} C_VEL
LIN {X 0,Y 504.27,Z 571.449,A -85,B 0,C 180,E1 23279.633,E2 23279.633} C_VEL
LIN {X 0,Y 505.643,Z 542.689,A -85,B 0,C 180,E1 23277.259,E2 23277.259} C_VEL
LIN {X 0,Y 498.78,Z 522.807,A -85,B 0,C 180,E1 23274.983,E2 23274.983} C_VEL
LIN {X 0,Y 496.79,Z 517.109,A -85,B 0,C 180,E1 23274.236,E2 23274.236} C_VEL
LIN {X 0,Y 496.76,Z 516.916,A -85,B 0,C 180,E1 23270.797,E2 23270.797} C_VEL
LIN {X 0,Y 496.726,Z 516.921,A -85,B 0,C 180,E1 23267.449,E2 23267.449} C_VEL
LIN {X 0,Y 496.76,Z 516.918,A -85,B 0,C 180,E1 23263.979,E2 23263.979} C_VEL
LIN {X 0,Y 496.757,Z 516.918,A -85,B 0,C 180,E1 23260.471,E2 23260.471} C_VEL
LIN {X 0,Y 496.714,Z 516.922,A -85,B 0,C 180,E1 23257.004,E2 23257.004} C_VEL
LIN {X 0,Y 496.731,Z 516.922,A -85,B 0,C 180,E1 23253.472,E2 23253.472} C_VEL
LIN {X 0,Y 496.776,Z 516.919,A -85,B 0,C 180,E1 23249.944,E2 23249.944} C_VEL
LIN {X 0,Y 496.707,Z 516.921,A -85,B 0,C 180,E1 23246.544,E2 23246.544} C_VEL
LIN {X 0,Y 496.706,Z 516.921,A -85,B 0,C 180,E1 23242.987,E2 23242.987} C_VEL
LIN {X 0,Y 496.756,Z 516.913,A -85,B 0,C 180,E1 23239.632,E2 23239.632} C_VEL
LIN {X 0,Y 496.696,Z 516.924,A -85,B 0,C 180,E1 23236.239,E2 23236.239} C_VEL
LIN {X 0,Y 496.692,Z 516.924,A -85,B 0,C 180,E1 23232.675,E2 23232.675} C_VEL
LIN {X 0,Y 496.747,Z 516.912,A -85,B 0,C 180,E1 23229.266,E2 23229.266} C_VEL
LIN {X 0,Y 496.693,Z 516.923,A -85,B 0,C 180,E1 23226.008,E2 23226.008} C_VEL
LIN {X 0,Y 496.701,Z 516.923,A -85,B 0,C 180,E1 23222.423,E2 23222.423} C_VEL
LIN {X 0,Y 496.764,Z 516.911,A -85,B 0,C 180,E1 23219.077,E2 23219.077} C_VEL
LIN {X 0,Y 496.711,Z 516.92,A -85,B 0,C 180,E1 23215.613,E2 23215.613} C_VEL
LIN {X 0,Y 496.712,Z 516.92,A -85,B 0,C 180,E1 23212.132,E2 23212.132} C_VEL
LIN {X 0,Y 496.768,Z 516.921,A -85,B 0,C 180,E1 23208.741,E2 23208.741} C_VEL
LIN {X 0,Y 496.723,Z 516.918,A -85,B 0,C 180,E1 23205.307,E2 23205.307} C_VEL
LIN {X 0,Y 496.722,Z 516.918,A -85,B 0,C 180,E1 23201.803,E2 23201.803} C_VEL
LIN {X 0,Y 496.774,Z 516.916,A -85,B 0,C 180,E1 23198.387,E2 23198.387} C_VEL
LIN {X 0,Y 496.745,Z 516.918,A -85,B 0,C 180,E1 23194.868,E2 23194.868} C_VEL
LIN {X 0,Y 496.727,Z 516.922,A -85,B 0,C 180,E1 23191.345,E2 23191.345} C_VEL
LIN {X 0,Y 496.764,Z 516.916,A -85,B 0,C 180,E1 23187.902,E2 23187.902} C_VEL
LIN {X 0,Y 496.766,Z 516.918,A -85,B 0,C 180,E1 23184.395,E2 23184.395} C_VEL
LIN {X 0,Y 496.79,Z 517.145,A -85,B 0,C 180,E1 23181.573,E2 23181.573} C_VEL
LIN {X 0,Y 501.613,Z 534.021,A -85,B 0,C 180,E1 23178.868,E2 23178.868} C_VEL
LIN {X 0,Y 502.53,Z 538.506,A -85,B 0,C 180,E1 23178.2,E2 23178.2} C_VEL
LIN {X 0,Y 501.041,Z 566.435,A -85,B 0,C 180,E1 23174.616,E2 23174.616} C_VEL
LIN {X 0,Y 499.753,Z 595.024,A -85,B 0,C 180,E1 23171.013,E2 23171.013} C_VEL
LIN {X 0,Y 498.584,Z 600.447,A -85,B 0,C 180,E1 23170.389,E2 23170.389} C_VEL
LIN {X 0,Y 491.836,Z 616.245,A -85,B 0,C 180,E1 23168.728,E2 23168.728} C_VEL
LIN {X 0,Y 491.161,Z 620.116,A -85,B 0,C 180,E1 23168.268,E2 23168.268} C_VEL
LIN {X 0,Y 490.789,Z 632.159,A -85,B 0,C 180,E1 23166.808,E2 23166.808} C_VEL
LIN {X 0,Y 493.034,Z 646.243,A -85,B 0,C 180,E1 23166.461,E2 23166.461} C_VEL
LIN {X 0,Y 492.008,Z 747.981,A -85,B 0,C 180,E1 23164.874,E2 23164.874} C_VEL
LIN {X 0,Y 491.754,Z 763.216,A -85,B 0,C 180,E1 23164.414,E2 23164.414} C_VEL
LIN {X 0,Y 491.34,Z 777.675,A -85,B 0,C 180,E1 23163.743,E2 23163.743} C_VEL
LIN {X 0,Y 490.862,Z 790.424,A -85,B 0,C 180,E1 23162.941,E2 23162.941} C_VEL
LIN {X 0,Y 490.277,Z 803.329,A -85,B 0,C 180,E1 23161.879,E2 23161.879} C_VEL
LIN {X 0,Y 489.765,Z 814.557,A -85,B 0,C 180,E1 23160.684,E2 23160.684} C_VEL
LIN {X 0,Y 489.298,Z 824.398,A -85,B 0,C 180,E1 23159.364,E2 23159.364} C_VEL
LIN {X 0,Y 488.872,Z 833.478,A -85,B 0,C 180,E1 23157.791,E2 23157.791} C_VEL
LIN {X 0,Y 488.589,Z 840.291,A -85,B 0,C 180,E1 23156.229,E2 23156.229} C_VEL
LIN {X 0,Y 488.412,Z 845.66,A -85,B 0,C 180,E1 23154.552,E2 23154.552} C_VEL
LIN {X 0,Y 488.304,Z 849.379,A -85,B 0,C 180,E1 23152.764,E2 23152.764} C_VEL
LIN {X 0,Y 488.249,Z 851.24,A -85,B 0,C 180,E1 23150.961,E2 23150.961} C_VEL
LIN {X 0,Y 488.242,Z 851.374,A -85,B 0,C 180,E1 23149.248,E2 23149.248} C_VEL
LIN {X 0,Y 488.274,Z 849.645,A -85,B 0,C 180,E1 23147.393,E2 23147.393} C_VEL
LIN {X 0,Y 488.36,Z 846.283,A -85,B 0,C 180,E1 23145.676,E2 23145.676} C_VEL
LIN {X 0,Y 488.521,Z 841.152,A -85,B 0,C 180,E1 23143.973,E2 23143.973} C_VEL
LIN {X 0,Y 488.784,Z 833.959,A -85,B 0,C 180,E1 23142.281,E2 23142.281} C_VEL
LIN {X 0,Y 489.136,Z 825.852,A -85,B 0,C 180,E1 23140.837,E2 23140.837} C_VEL
LIN {X 0,Y 489.597,Z 816.034,A -85,B 0,C 180,E1 23139.462,E2 23139.462} C_VEL
LIN {X 0,Y 490.142,Z 803.935,A -85,B 0,C 180,E1 23138.148,E2 23138.148} C_VEL
LIN {X 0,Y 490.687,Z 791.286,A -85,B 0,C 180,E1 23137.09,E2 23137.09} C_VEL
LIN {X 0,Y 491.178,Z 778.223,A -85,B 0,C 180,E1 23136.25,E2 23136.25} C_VEL
LIN {X 0,Y 491.621,Z 763.012,A -85,B 0,C 180,E1 23135.542,E2 23135.542} C_VEL
LIN {X 0,Y 491.894,Z 747.358,A -85,B 0,C 180,E1 23135.074,E2 23135.074} C_VEL
LIN {X 0,Y 492.597,Z 643.363,A -85,B 0,C 180,E1 23133.464,E2 23133.464} C_VEL
LIN {X 0,Y 490.635,Z 632.152,A -85,B 0,C 180,E1 23133.185,E2 23133.185} C_VEL
LIN {X 0,Y 491.618,Z 604.388,A -85,B 0,C 180,E1 23129.766,E2 23129.766} C_VEL
LIN {X 0,Y 492.938,Z 574.919,A -85,B 0,C 180,E1 23126.044,E2 23126.044} C_VEL
LIN {X 0,Y 494.415,Z 545.978,A -85,B 0,C 180,E1 23122.329,E2 23122.329} C_VEL
LIN {X 0,Y 494.513,Z 538.825,A -85,B 0,C 180,E1 23121.386,E2 23121.386} C_VEL
LIN {X 0,Y 489.374,Z 520.211,A -85,B 0,C 180,E1 23118.509,E2 23118.509} C_VEL
LIN {X 0,Y 488.781,Z 517.991,A -85,B 0,C 180,E1 23118.093,E2 23118.093} C_VEL
LIN {X 0,Y 488.754,Z 517.913,A -85,B 0,C 180,E1 23114.577,E2 23114.577} C_VEL
LIN {X 0,Y 488.803,Z 517.909,A -85,B 0,C 180,E1 23111.144,E2 23111.144} C_VEL
LIN {X 0,Y 488.766,Z 517.906,A -85,B 0,C 180,E1 23107.763,E2 23107.763} C_VEL
LIN {X 0,Y 488.749,Z 517.912,A -85,B 0,C 180,E1 23104.298,E2 23104.298} C_VEL
LIN {X 0,Y 488.799,Z 517.889,A -85,B 0,C 180,E1 23100.863,E2 23100.863} C_VEL
LIN {X 0,Y 488.761,Z 517.899,A -85,B 0,C 180,E1 23097.441,E2 23097.441} C_VEL
LIN {X 0,Y 488.748,Z 517.91,A -85,B 0,C 180,E1 23093.903,E2 23093.903} C_VEL
LIN {X 0,Y 488.794,Z 517.912,A -85,B 0,C 180,E1 23090.46,E2 23090.46} C_VEL
LIN {X 0,Y 488.76,Z 517.902,A -85,B 0,C 180,E1 23087.224,E2 23087.224} C_VEL
LIN {X 0,Y 488.757,Z 517.911,A -85,B 0,C 180,E1 23083.746,E2 23083.746} C_VEL
LIN {X 0,Y 488.812,Z 517.901,A -85,B 0,C 180,E1 23080.269,E2 23080.269} C_VEL
LIN {X 0,Y 488.773,Z 517.912,A -85,B 0,C 180,E1 23076.826,E2 23076.826} C_VEL
LIN {X 0,Y 488.759,Z 517.9,A -85,B 0,C 180,E1 23073.388,E2 23073.388} C_VEL
LIN {X 0,Y 488.816,Z 517.909,A -85,B 0,C 180,E1 23069.941,E2 23069.941} C_VEL
LIN {X 0,Y 488.779,Z 517.898,A -85,B 0,C 180,E1 23066.484,E2 23066.484} C_VEL
LIN {X 0,Y 488.764,Z 517.909,A -85,B 0,C 180,E1 23063,E2 23063} C_VEL
LIN {X 0,Y 488.816,Z 517.898,A -85,B 0,C 180,E1 23059.601,E2 23059.601} C_VEL
LIN {X 0,Y 488.783,Z 517.897,A -85,B 0,C 180,E1 23056.153,E2 23056.153} C_VEL
LIN {X 0,Y 488.768,Z 517.909,A -85,B 0,C 180,E1 23052.644,E2 23052.644} C_VEL
LIN {X 0,Y 488.808,Z 517.887,A -85,B 0,C 180,E1 23049.181,E2 23049.181} C_VEL
LIN {X 0,Y 488.787,Z 517.906,A -85,B 0,C 180,E1 23045.871,E2 23045.871} C_VEL
LIN {X 0,Y 488.773,Z 517.903,A -85,B 0,C 180,E1 23042.345,E2 23042.345} C_VEL
LIN {X 0,Y 488.822,Z 517.901,A -85,B 0,C 180,E1 23038.945,E2 23038.945} C_VEL
LIN {X 0,Y 488.802,Z 517.911,A -85,B 0,C 180,E1 23035.425,E2 23035.425} C_VEL
LIN {X 0,Y 488.776,Z 517.894,A -85,B 0,C 180,E1 23032.004,E2 23032.004} C_VEL
LIN {X 0,Y 488.818,Z 517.906,A -85,B 0,C 180,E1 23028.556,E2 23028.556} C_VEL
LIN {X 0,Y 488.811,Z 517.897,A -85,B 0,C 180,E1 23025.065,E2 23025.065} C_VEL
LIN {X 0,Y 488.782,Z 517.909,A -85,B 0,C 180,E1 23021.638,E2 23021.638} C_VEL
LIN {X 0,Y 488.817,Z 517.902,A -85,B 0,C 180,E1 23018.144,E2 23018.144} C_VEL
LIN {X 0,Y 488.819,Z 517.906,A -85,B 0,C 180,E1 23014.691,E2 23014.691} C_VEL
LIN {X 0,Y 488.785,Z 517.909,A -85,B 0,C 180,E1 23011.268,E2 23011.268} C_VEL
LIN {X 0,Y 488.821,Z 517.904,A -85,B 0,C 180,E1 23007.862,E2 23007.862} C_VEL
LIN {X 0,Y 488.828,Z 517.903,A -85,B 0,C 180,E1 23004.29,E2 23004.29} C_VEL
LIN {X 0,Y 488.792,Z 517.905,A -85,B 0,C 180,E1 23000.796,E2 23000.796} C_VEL
LIN {X 0,Y 488.802,Z 517.907,A -85,B 0,C 180,E1 22997.226,E2 22997.226} C_VEL
LIN {X 0,Y 488.834,Z 517.908,A -85,B 0,C 180,E1 22993.734,E2 22993.734} C_VEL
LIN {X 0,Y 488.804,Z 517.907,A -85,B 0,C 180,E1 22990.267,E2 22990.267} C_VEL
LIN {X 0,Y 488.797,Z 517.908,A -85,B 0,C 180,E1 22986.675,E2 22986.675} C_VEL
LIN {X 0,Y 488.874,Z 518.348,A -85,B 0,C 180,E1 22986.123,E2 22986.123} C_VEL
LIN {X 0,Y 497.44,Z 542.782,A -85,B 0,C 180,E1 22983.278,E2 22983.278} C_VEL
LIN {X 0,Y 498.41,Z 545.989,A -85,B 0,C 180,E1 22982.931,E2 22982.931} C_VEL
LIN {X 0,Y 496.089,Z 590.463,A -85,B 0,C 180,E1 22979.258,E2 22979.258} C_VEL
LIN {X 0,Y 495.008,Z 615.653,A -85,B 0,C 180,E1 22977.246,E2 22977.246} C_VEL
LIN {X 0,Y 496.997,Z 632.02,A -85,B 0,C 180,E1 22976.895,E2 22976.895} C_VEL
LIN {X 0,Y 495.304,Z 821.713,A -85,B 0,C 180,E1 22974.088,E2 22974.088} C_VEL
LIN {X 0,Y 494.74,Z 840.601,A -85,B 0,C 180,E1 22973.6,E2 22973.6} C_VEL
LIN {X 0,Y 494.043,Z 859.175,A -85,B 0,C 180,E1 22972.9,E2 22972.9} C_VEL
LIN {X 0,Y 493.279,Z 876.664,A -85,B 0,C 180,E1 22972.023,E2 22972.023} C_VEL
LIN {X 0,Y 492.372,Z 893.765,A -85,B 0,C 180,E1 22970.94,E2 22970.94} C_VEL
LIN {X 0,Y 491.523,Z 909.991,A -85,B 0,C 180,E1 22969.673,E2 22969.673} C_VEL
LIN {X 0,Y 490.651,Z 925.857,A -85,B 0,C 180,E1 22968.167,E2 22968.167} C_VEL
LIN {X 0,Y 489.907,Z 939.556,A -85,B 0,C 180,E1 22966.602,E2 22966.602} C_VEL
LIN {X 0,Y 489.256,Z 952.704,A -85,B 0,C 180,E1 22964.801,E2 22964.801} C_VEL
LIN {X 0,Y 488.759,Z 963.581,A -85,B 0,C 180,E1 22963.005,E2 22963.005} C_VEL
LIN {X 0,Y 488.403,Z 973.122,A -85,B 0,C 180,E1 22961.096,E2 22961.096} C_VEL
LIN {X 0,Y 488.147,Z 981.247,A -85,B 0,C 180,E1 22959.075,E2 22959.075} C_VEL
LIN {X 0,Y 487.998,Z 987.861,A -85,B 0,C 180,E1 22956.944,E2 22956.944} C_VEL
LIN {X 0,Y 487.931,Z 992.6,A -85,B 0,C 180,E1 22954.82,E2 22954.82} C_VEL
LIN {X 0,Y 487.911,Z 995.552,A -85,B 0,C 180,E1 22952.703,E2 22952.703} C_VEL
LIN {X 0,Y 487.908,Z 996.839,A -85,B 0,C 180,E1 22950.471,E2 22950.471} C_VEL
LIN {X 0,Y 487.912,Z 996.319,A -85,B 0,C 180,E1 22948.24,E2 22948.24} C_VEL
LIN {X 0,Y 487.921,Z 994.131,A -85,B 0,C 180,E1 22946.124,E2 22946.124} C_VEL
LIN {X 0,Y 487.958,Z 990.193,A -85,B 0,C 180,E1 22944.003,E2 22944.003} C_VEL
LIN {X 0,Y 488.065,Z 984.424,A -85,B 0,C 180,E1 22941.876,E2 22941.876} C_VEL
LIN {X 0,Y 488.29,Z 976.688,A -85,B 0,C 180,E1 22939.74,E2 22939.74} C_VEL
LIN {X 0,Y 488.609,Z 967.355,A -85,B 0,C 180,E1 22937.715,E2 22937.715} C_VEL
LIN {X 0,Y 489.071,Z 956.498,A -85,B 0,C 180,E1 22935.802,E2 22935.802} C_VEL
LIN {X 0,Y 489.664,Z 944.136,A -85,B 0,C 180,E1 22934.002,E2 22934.002} C_VEL
LIN {X 0,Y 490.394,Z 930.222,A -85,B 0,C 180,E1 22932.317,E2 22932.317} C_VEL
LIN {X 0,Y 491.212,Z 915.311,A -85,B 0,C 180,E1 22930.816,E2 22930.816} C_VEL
LIN {X 0,Y 492.048,Z 899.341,A -85,B 0,C 180,E1 22929.484,E2 22929.484} C_VEL
LIN {X 0,Y 492.965,Z 881.842,A -85,B 0,C 180,E1 22928.299,E2 22928.299} C_VEL
LIN {X 0,Y 493.784,Z 864.07,A -85,B 0,C 180,E1 22927.345,E2 22927.345} C_VEL
LIN {X 0,Y 494.514,Z 845.657,A -85,B 0,C 180,E1 22926.592,E2 22926.592} C_VEL
LIN {X 0,Y 495.1,Z 827.034,A -85,B 0,C 180,E1 22926.052,E2 22926.052} C_VEL
LIN {X 0,Y 495.448,Z 805.567,A -85,B 0,C 180,E1 22925.671,E2 22925.671} C_VEL
LIN {X 0,Y 496.728,Z 629.042,A -85,B 0,C 180,E1 22923.08,E2 22923.08} C_VEL
LIN {X 0,Y 494.933,Z 615.519,A -85,B 0,C 180,E1 22922.774,E2 22922.774} C_VEL
LIN {X 0,Y 497.007,Z 570.695,A -85,B 0,C 180,E1 22919.141,E2 22919.141} C_VEL
LIN {X 0,Y 498.326,Z 545.358,A -85,B 0,C 180,E1 22917.002,E2 22917.002} C_VEL
LIN {X 0,Y 491.639,Z 525.988,A -85,B 0,C 180,E1 22914.725,E2 22914.725} C_VEL
LIN {X 0,Y 488.824,Z 518.116,A -85,B 0,C 180,E1 22913.687,E2 22913.687} C_VEL
LIN {X 0,Y 488.833,Z 517.908,A -85,B 0,C 180,E1 22910.27,E2 22910.27} C_VEL
LIN {X 0,Y 488.811,Z 517.905,A -85,B 0,C 180,E1 22906.735,E2 22906.735} C_VEL
LIN {X 0,Y 488.783,Z 517.912,A -85,B 0,C 180,E1 22903.257,E2 22903.257} C_VEL
LIN {X 0,Y 488.805,Z 517.907,A -85,B 0,C 180,E1 22899.734,E2 22899.734} C_VEL
LIN {X 0,Y 488.819,Z 517.907,A -85,B 0,C 180,E1 22896.238,E2 22896.238} C_VEL
LIN {X 0,Y 488.773,Z 517.909,A -85,B 0,C 180,E1 22892.79,E2 22892.79} C_VEL
LIN {X 0,Y 488.774,Z 517.908,A -85,B 0,C 180,E1 22889.145,E2 22889.145} C_VEL
LIN {X 0,Y 488.822,Z 517.911,A -85,B 0,C 180,E1 22885.698,E2 22885.698} C_VEL
LIN {X 0,Y 488.773,Z 517.909,A -85,B 0,C 180,E1 22882.237,E2 22882.237} C_VEL
LIN {X 0,Y 488.756,Z 517.906,A -85,B 0,C 180,E1 22878.727,E2 22878.727} C_VEL
LIN {X 0,Y 488.801,Z 517.901,A -85,B 0,C 180,E1 22875.3,E2 22875.3} C_VEL
LIN {X 0,Y 488.765,Z 517.913,A -85,B 0,C 180,E1 22871.924,E2 22871.924} C_VEL
LIN {X 0,Y 488.749,Z 517.91,A -85,B 0,C 180,E1 22868.47,E2 22868.47} C_VEL
LIN {X 0,Y 488.81,Z 517.899,A -85,B 0,C 180,E1 22865.097,E2 22865.097} C_VEL
LIN {X 0,Y 488.773,Z 517.913,A -85,B 0,C 180,E1 22861.641,E2 22861.641} C_VEL
LIN {X 0,Y 488.761,Z 517.911,A -85,B 0,C 180,E1 22858.124,E2 22858.124} C_VEL
LIN {X 0,Y 488.811,Z 517.901,A -85,B 0,C 180,E1 22854.718,E2 22854.718} C_VEL
LIN {X 0,Y 488.79,Z 517.908,A -85,B 0,C 180,E1 22851.293,E2 22851.293} C_VEL
LIN {X 0,Y 488.773,Z 517.91,A -85,B 0,C 180,E1 22847.836,E2 22847.836} C_VEL
LIN {X 0,Y 488.813,Z 517.908,A -85,B 0,C 180,E1 22844.335,E2 22844.335} C_VEL
LIN {X 0,Y 488.823,Z 517.911,A -85,B 0,C 180,E1 22840.772,E2 22840.772} C_VEL
LIN {X 0,Y 488.786,Z 517.912,A -85,B 0,C 180,E1 22837.255,E2 22837.255} C_VEL
LIN {X 0,Y 488.792,Z 517.908,A -85,B 0,C 180,E1 22833.619,E2 22833.619} C_VEL
LIN {X 0,Y 488.837,Z 517.903,A -85,B 0,C 180,E1 22830.128,E2 22830.128} C_VEL
LIN {X 0,Y 488.822,Z 517.909,A -85,B 0,C 180,E1 22826.558,E2 22826.558} C_VEL
LIN {X 0,Y 488.798,Z 517.913,A -85,B 0,C 180,E1 22823.03,E2 22823.03} C_VEL
LIN {X 0,Y 488.877,Z 518.209,A -85,B 0,C 180,E1 22822.078,E2 22822.078} C_VEL
LIN {X 0,Y 493.768,Z 535.109,A -85,B 0,C 180,E1 22819.304,E2 22819.304} C_VEL
LIN {X 0,Y 495.125,Z 540.682,A -85,B 0,C 180,E1 22818.442,E2 22818.442} C_VEL
LIN {X 0,Y 493.517,Z 568.354,A -85,B 0,C 180,E1 22814.838,E2 22814.838} C_VEL
LIN {X 0,Y 492.06,Z 598.32,A -85,B 0,C 180,E1 22811.014,E2 22811.014} C_VEL
LIN {X 0,Y 491.161,Z 620.116,A -85,B 0,C 180,E1 22808.268,E2 22808.268} C_VEL
LIN {X 0,Y 490.097,Z 623.992,A -85,B 0,C 180,E1 22807.85,E2 22807.85} C_VEL
LIN {X 0,Y 486.714,Z 630.638,A -85,B 0,C 180,E1 22807.356,E2 22807.356} C_VEL
LIN {X 0,Y 484.796,Z 636.022,A -85,B 0,C 180,E1 22807.1,E2 22807.1} C_VEL
LIN {X 0,Y 484.66,Z 640.368,A -85,B 0,C 180,E1 22806.962,E2 22806.962} C_VEL
LIN {X 0,Y 485.618,Z 647.936,A -85,B 0,C 180,E1 22806.795,E2 22806.795} C_VEL
LIN {X 0,Y 484.507,Z 748.569,A -85,B 0,C 180,E1 22805.193,E2 22805.193} C_VEL
LIN {X 0,Y 484.236,Z 763.592,A -85,B 0,C 180,E1 22804.734,E2 22804.734} C_VEL
LIN {X 0,Y 483.793,Z 778.113,A -85,B 0,C 180,E1 22804.056,E2 22804.056} C_VEL
LIN {X 0,Y 483.28,Z 790.961,A -85,B 0,C 180,E1 22803.243,E2 22803.243} C_VEL
LIN {X 0,Y 482.639,Z 803.929,A -85,B 0,C 180,E1 22802.164,E2 22802.164} C_VEL
LIN {X 0,Y 482.073,Z 815.25,A -85,B 0,C 180,E1 22800.951,E2 22800.951} C_VEL
LIN {X 0,Y 481.558,Z 825.174,A -85,B 0,C 180,E1 22799.61,E2 22799.61} C_VEL
LIN {X 0,Y 481.075,Z 834.318,A -85,B 0,C 180,E1 22798.011,E2 22798.011} C_VEL
LIN {X 0,Y 480.751,Z 841.214,A -85,B 0,C 180,E1 22796.424,E2 22796.424} C_VEL
LIN {X 0,Y 480.542,Z 846.658,A -85,B 0,C 180,E1 22794.718,E2 22794.718} C_VEL
LIN {X 0,Y 480.407,Z 850.435,A -85,B 0,C 180,E1 22792.901,E2 22792.901} C_VEL
LIN {X 0,Y 480.34,Z 852.361,A -85,B 0,C 180,E1 22791.104,E2 22791.104} C_VEL
LIN {X 0,Y 480.329,Z 852.533,A -85,B 0,C 180,E1 22789.198,E2 22789.198} C_VEL
LIN {X 0,Y 480.37,Z 850.772,A -85,B 0,C 180,E1 22787.313,E2 22787.313} C_VEL
LIN {X 0,Y 480.474,Z 847.274,A -85,B 0,C 180,E1 22785.527,E2 22785.527} C_VEL
LIN {X 0,Y 480.658,Z 842.222,A -85,B 0,C 180,E1 22783.838,E2 22783.838} C_VEL
LIN {X 0,Y 480.958,Z 835.01,A -85,B 0,C 180,E1 22782.118,E2 22782.118} C_VEL
LIN {X 0,Y 481.351,Z 826.893,A -85,B 0,C 180,E1 22780.651,E2 22780.651} C_VEL
LIN {X 0,Y 481.832,Z 817.524,A -85,B 0,C 180,E1 22779.313,E2 22779.313} C_VEL
LIN {X 0,Y 482.39,Z 806.186,A -85,B 0,C 180,E1 22778.04,E2 22778.04} C_VEL
LIN {X 0,Y 482.941,Z 794.621,A -85,B 0,C 180,E1 22777.014,E2 22777.014} C_VEL
LIN {X 0,Y 483.528,Z 780.427,A -85,B 0,C 180,E1 22776.052,E2 22776.052} C_VEL
LIN {X 0,Y 483.974,Z 766.497,A -85,B 0,C 180,E1 22775.362,E2 22775.362} C_VEL
LIN {X 0,Y 484.303,Z 751.603,A -85,B 0,C 180,E1 22774.857,E2 22774.857} C_VEL
LIN {X 0,Y 484.523,Z 730.078,A -85,B 0,C 180,E1 22774.462,E2 22774.462} C_VEL
LIN {X 0,Y 485.13,Z 644.319,A -85,B 0,C 180,E1 22773.137,E2 22773.137} C_VEL
LIN {X 0,Y 482.926,Z 631.885,A -85,B 0,C 180,E1 22772.817,E2 22772.817} C_VEL
LIN {X 0,Y 484.024,Z 603.693,A -85,B 0,C 180,E1 22769.288,E2 22769.288} C_VEL
LIN {X 0,Y 485.427,Z 575.094,A -85,B 0,C 180,E1 22765.628,E2 22765.628} C_VEL
LIN {X 0,Y 487.013,Z 546.065,A -85,B 0,C 180,E1 22761.855,E2 22761.855} C_VEL
LIN {X 0,Y 487.099,Z 541.645,A -85,B 0,C 180,E1 22761.262,E2 22761.262} C_VEL
LIN {X 0,Y 482.042,Z 523.31,A -85,B 0,C 180,E1 22758.392,E2 22758.392} C_VEL
LIN {X 0,Y 480.882,Z 518.969,A -85,B 0,C 180,E1 22757.633,E2 22757.633} C_VEL
LIN {X 0,Y 480.817,Z 518.903,A -85,B 0,C 180,E1 22754.192,E2 22754.192} C_VEL
LIN {X 0,Y 480.817,Z 518.899,A -85,B 0,C 180,E1 22750.566,E2 22750.566} C_VEL
LIN {X 0,Y 480.866,Z 518.873,A -85,B 0,C 180,E1 22747.092,E2 22747.092} C_VEL
LIN {X 0,Y 480.831,Z 518.9,A -85,B 0,C 180,E1 22743.578,E2 22743.578} C_VEL
LIN {X 0,Y 480.804,Z 518.875,A -85,B 0,C 180,E1 22740.061,E2 22740.061} C_VEL
LIN {X 0,Y 480.842,Z 518.9,A -85,B 0,C 180,E1 22736.563,E2 22736.563} C_VEL
LIN {X 0,Y 480.848,Z 518.894,A -85,B 0,C 180,E1 22733.065,E2 22733.065} C_VEL
LIN {X 0,Y 480.811,Z 518.902,A -85,B 0,C 180,E1 22729.707,E2 22729.707} C_VEL
LIN {X 0,Y 480.857,Z 518.895,A -85,B 0,C 180,E1 22726.346,E2 22726.346} C_VEL
LIN {X 0,Y 480.845,Z 518.901,A -85,B 0,C 180,E1 22722.841,E2 22722.841} C_VEL
LIN {X 0,Y 480.816,Z 518.897,A -85,B 0,C 180,E1 22719.365,E2 22719.365} C_VEL
LIN {X 0,Y 480.85,Z 518.892,A -85,B 0,C 180,E1 22715.901,E2 22715.901} C_VEL
LIN {X 0,Y 480.859,Z 518.889,A -85,B 0,C 180,E1 22712.419,E2 22712.419} C_VEL
LIN {X 0,Y 480.821,Z 518.899,A -85,B 0,C 180,E1 22708.981,E2 22708.981} C_VEL
LIN {X 0,Y 480.845,Z 518.887,A -85,B 0,C 180,E1 22705.495,E2 22705.495} C_VEL
LIN {X 0,Y 480.882,Z 518.9,A -85,B 0,C 180,E1 22701.979,E2 22701.979} C_VEL
LIN {X 0,Y 480.828,Z 518.888,A -85,B 0,C 180,E1 22698.527,E2 22698.527} C_VEL
